// TwinCAT 3 PLC project MQPLC
// Title: YK_RFH
// Company: YK
// Author: SJ
// ProjectVersion: V1.1
// ProgramVersion: 3.1.4024.0
// CompilerDefines: VISU_USEWSTRING
// libraries:
//   Lib_Basic, * (Beckhoff_GZ)
//   Lib_FileOperation, * (Beckhoff_GZ)
//   Tc2_EtherCAT, * (Beckhoff Automation GmbH)
//   Tc2_Math, * (Beckhoff Automation GmbH)
//   Tc2_MC2, * (Beckhoff Automation GmbH)
//   Tc2_MC2_Camming, * (Beckhoff Automation GmbH)
//   Tc2_MC2_FlyingSaw, * (Beckhoff Automation GmbH)
//   Tc2_Standard, * (Beckhoff Automation GmbH)
//   Tc2_System, * (Beckhoff Automation GmbH)
//   Tc2_TcpIp, * (Beckhoff Automation GmbH)
//   Tc2_Utilities, * (Beckhoff Automation GmbH)
//   Tc2_XmlDataSrv, * (Beckhoff Automation GmbH)
//   Tc3_MC2_AdvancedHoming, * (Beckhoff Automation GmbH)
//   Tc3_Module, * (Beckhoff Automation GmbH)
//   VisuDialogs, * (System)
//   VisuElemEventTable, * (System)
//   VisuSymbols, * (System)
//   VisuSymbols,3.5.10.0,System
// project tree:
//   DUTs/01_AxisCO_Ntrol/ ST_ECYCtrl.TcDUT, ST_JXCE.TcDUT, ST_DustMotor.TcDUT, MC_AxisParameter.TcDUT, ST_SetpMotor.TcDUT
//   DUTs/01_AxisCO_Ntrol_1/ ST_AxisCmd.TcDUT, ST_AxisCtrl.TcDUT, ST_AxisIo.TcDUT, ST_AxisStatus.TcDUT, ST_Axis_Par.TcDUT
//   DUTs/02_Cylinder/ ST_CyCmd.TcDUT, ST_CyCtrl.TcDUT, ST_CYIo.TcDUT, ST_CyStatus.TcDUT
//   DUTs/04_Rectify/ ST_RecCtrl.TcDUT, ST_RecCmd.TcDUT, ST_RecIo.TcDUT, ST_RecStatus.TcDUT
//   DUTs/06_Interface/FB_Interface/ ST_Cam.TcDUT, ST_Gear.TcDUT, ST_GearInPos.TcDUT, ST_RecY.TcDUT, ST_TenBuffer.TcDUT, ST_Tension_1.TcDUT, ST_Tension.TcDUT
//   DUTs/06_Interface/Method/ ST_Method.TcDUT, ST_MethodOut.TcDUT
//   DUTs/07_Name/ ST_MotorName.TcDUT, ST_NGMark.TcDUT, ST_TableNo.TcDUT, ST_CylinderName.TcDUT, ST_VirAxisName.TcDUT, ST_AxisName.TcDUT, ST_RecName.TcDUT, ST_ElectValveName.TcDUT
//   DUTs/09_保持型汇总/ LocalProduction.TcDUT, ST_Data.TcDUT, ST_Name.TcDUT, ST_Parameter.TcDUT
//   DUTs/30_Parameter/ ST_DT_To_MQ_MES.TcDUT, ST_MouldRecY.TcDUT, ST_MQ_To_DT_MES.TcDUT, ST_ParFilterAD.TcDUT, ST_ParFilterDA.TcDUT, ST_ParMachine.TcDUT, ST_MoQiePar.TcDUT, ST_ParProduct.TcDUT, ST_ParPublic.TcDUT, ST_ParTemperature.TcDUT
//   DUTs/31_其他辅助/ ST_Timedata_2.TcDUT, File_com_typ.TcDUT, ST_DATA_NEED_BE_PERSIS.TcDUT
//   DUTs/32_系统/ ST_SystemPart.TcDUT, IModeEN.TcDUT, IRecipe.TcDUT, ST_SysCmd.TcDUT, ST_SystemPublic.TcDUT
//   DUTs/33_M2/ ST_BeltData.TcDUT, ST_TabData.TcDUT, ST_AlarmWarn.TcDUT, ST_BeltNo.TcDUT, ST_IntervalData.TcDUT, ST_IntervalNo.TcDUT, ST_TabNo.TcDUT
//   DUTs/34_M1/ ST_CCDio.TcDUT, ST_Rectify.TcDUT
//   DUTs/35_CCD/ ST_CCDComCuter.TcDUT, ST_CCDComLineScan.TcDUT, ST_CCDComR_Mould.TcDUT, ST_CCDComSize.TcDUT, ST_CCDCom.TcDUT, STCcdData.TcDUT, STCcdDataSend.TcDUT
//   DUTs/38_交互/ DToM_Process.TcDUT, DToM_System.TcDUT, MToD_Process.TcDUT, MToD_System.TcDUT, ST_P2InteractPart.TcDUT, ST_P2InteractPub.TcDUT
//   DUTs/39_记忆/ ST_Meney_Type.TcDUT
//   DUTs/MES/ DTM_Mes1.TcDUT, MTD_Mes1.TcDUT
//   DUTs/指纹/ ST_FingerprintKey.TcDUT
//   GVLs/ GVL_Par.TcGVL, GVL_Rectify.TcGVL, GVL_User2.TcGVL, GVL_User3.TcGVL, GCylinder.TcGVL, IO.TcGVL, GMotion.TcGVL, N.TcGVL, System.TcGVL, User01.TcGVL
//   POUs/BasicFunction/Basic/01_IO/ FB_Filter_AD.TcPOU (encrypted, skipped), FB_Filter_ADV2.TcPOU, FB_RotateSwitchCode.TcPOU (encrypted, skipped)
//   POUs/BasicFunction/Basic/02_Temperature/ FB_Blink.TcPOU (encrypted, skipped), FB_PulsPercentage.TcPOU (encrypted, skipped)
//   POUs/BasicFunction/Basic/03_Motion/ CS_AxisCtrl.TcPOU (encrypted, skipped)
//   POUs/BasicFunction/Basic/04_Gear/ FB_GearInDyn.TcPOU (encrypted, skipped), FB_GearInMulti.TcPOU (encrypted, skipped), FB_GearInPos.TcPOU (encrypted, skipped)
//   POUs/BasicFunction/Basic/05_Actuators/ FB_CylinderV2.TcPOU
//   POUs/BasicFunction/Basic/06_Public/ FC_AngleToLength.TcPOU (encrypted, skipped), FC_LengthToAngle.TcPOU (encrypted, skipped), f_Length2.TcPOU (encrypted, skipped), f_Length2_1.TcPOU (encrypted, skipped), PulseCtrl.TcPOU (encrypted, skipped), PulseGeneratorCtrl.TcPOU (encrypted, skipped)
//   POUs/BasicFunction/Basic/07_Ten/ FB_TensionBuffer.TcPOU (encrypted, skipped), FB_TensionPole.TcPOU, FB_TensionV3.TcPOU (encrypted, skipped), FB_TensionVirDriver.TcPOU
//   POUs/BasicFunction/Data/ Day_date.TcPOU, FB_DataTime.TcPOU, FB_ProductionDataLocal.TcPOU, FC_Filter_AA.TcPOU, FC_Variance.TcPOU, ScaleTrans.TcPOU, CS_Data.TcPOU, CS_Data_Test.TcPOU, CS_Recipe.TcPOU
//   POUs/BasicFunction/Motion/ Ax_FindHomeV3.TcPOU (encrypted, skipped), CS_DustMoter.TcPOU, FB_Electric_CY.TcPOU, FB_RectifyGM.TcPOU (encrypted, skipped), FB_TailCurl_PID.TcPOU, MS_Alarm.TcPOU, CS_SetpMoter.TcPOU
//   POUs/BasicFunction/User1/ FB_CamMQBeltV1.TcPOU (encrypted, skipped), FB_CamMQCCDPressV1.TcPOU (encrypted, skipped), FB_CamMQDriverV1.TcPOU (encrypted, skipped), FB_CamMQPushV1.TcPOU (encrypted, skipped), FB_CamMQPushV2.TcPOU (encrypted, skipped), FB_CamPoleBuffer.TcPOU (encrypted, skipped), FB_CamPoleBufferV2.TcPOU (encrypted, skipped), FB_CamPoleBuffer_1.TcPOU (encrypted, skipped), FB_CamPoleBuffer_BAK.TcPOU (encrypted, skipped), FB_CamVirDriver.TcPOU (encrypted, skipped), FB_CCD_Rounde.TcPOU, FB_DataXML.TcPOU, FB_DataXML_Old.TcPOU, FB_Rectify.TcPOU (encrypted, skipped), FB_TensionPole_1.TcPOU (encrypted, skipped)
//   POUs/BasicFunction/XFC/ FB_EL1259_IN.TcPOU, FB_TouchProbe_Ear.TcPOU
//   DUTs/08_IO/ ST_MoQieSenser.TcDUT, ST_MoQieButton.TcDUT
//   DUTs/06_Interface/ IData.TcDUT, IM2Glue.TcDUT
//   DUTs/36_ShortTest/ CMD.TcDUT, IShortTest.TcDUT, ShortDataShow.TcDUT, ShortPar.TcDUT
//   DUTs/37_Code/ ICode.TcDUT
//   POUs/BasicFunction/MES/ CS_CcdTcp.TcPOU, CS_CcdTcp_V2.TcPOU, CS_CodeTcp.TcPOU
//   POUs/BasicFunction/SystemInfo/ SystemInfoCtrl.TcPOU, TaskInfoCtrl.TcPOU
//   POUs/POUs/ AnPart.TcPOU, CaPart.TcPOU, FB_UserMain.TcPOU, FingerprintKey.TcPOU, IOLink.TcPOU, MAIN.TcPOU, MainState.TcPOU, ProductLocal.TcPOU
//   / Task_P1.TcTTO
// (motion and I/O tree: see PLC project dpplc)
// real-time tasks:
//   TASK Task P1: cycle T#2ms, priority 8, ADS port 350
//   TASK Task P2M1: cycle T#2ms, priority 16, ADS port 351
//   TASK Task P3: cycle T#2ms, priority 18, ADS port 352
//   TASK Task P2M2: cycle T#2ms, priority 14, ADS port 353
//   TASK Task P2M3: cycle T#2ms, priority 12, ADS port 354
//   TASK Task P2Main: cycle T#2ms, priority 10, ADS port 355
// variable links:
//   DPPLC/DPPLC Instance <-> MQPLC/MQPLC Instance
//     Task_P2M3 Inputs/IO.M_Pro <-> Task_P1 Outputs/IO.M_Pro
//     Task_P2M3 Outputs/IO.D_Pro <-> Task_P1 Inputs/IO.D_Pro
//     Task_P2M3 Outputs/IO.D_Sys/P3ReadParDone <-> Task_P1 Inputs/IO.D_Sys/P3ReadParDone
//     Task_P2M3 Outputs/IO.D_Sys/P3SaveParDone <-> Task_P1 Inputs/IO.D_Sys/P3SaveParDone
//     Task_P2M3 Outputs/IO.D_Sys/bP2ClearDo <-> Task_P1 Inputs/IO.D_Sys/bP2ClearDo
//     Task_P2M3 Outputs/IO.D_Sys/bP2ClearDone <-> Task_P1 Inputs/IO.D_Sys/bP2ClearDone
//     Task_P2M3 Outputs/IO.D_Sys/bP2Estop <-> Task_P1 Inputs/IO.D_Sys/bP2Estop
//     Task_P2M3 Outputs/IO.D_Sys/bP2M1Enable <-> Task_P1 Inputs/IO.D_Sys/bP2M1Enable
//     Task_P2M3 Outputs/IO.D_Sys/bP2M2Enable <-> Task_P1 Inputs/IO.D_Sys/bP2M2Enable
//     Task_P2M3 Outputs/IO.D_Sys/bP2M3Enable <-> Task_P1 Inputs/IO.D_Sys/bP2M3Enable
//     Task_P2M3 Outputs/IO.D_Sys/bP2Runing <-> Task_P1 Inputs/IO.D_Sys/bP2Runing
//     Task_P2M3 Outputs/IO.D_Sys/bP2Start <-> Task_P1 Inputs/IO.D_Sys/bP2Start
//     Task_P2M3 Outputs/IO.D_Sys/fM1MainSetPos <-> Task_P1 Inputs/IO.D_Sys/fM1MainSetPos
//     Task_P2M3 Outputs/IO.D_Sys/fM2MainSetPos <-> Task_P1 Inputs/IO.D_Sys/fM2MainSetPos
//     Task_P2M3 Outputs/IO.D_Sys/fM3MainSetPos <-> Task_P1 Inputs/IO.D_Sys/fM3MainSetPos
//     Task_P2M3 Outputs/IO.D_Sys/iAn1Ask <-> Task_P1 Inputs/IO.D_Sys/iAn1Ask
//     Task_P2M3 Outputs/IO.D_Sys/iAn2Ask <-> Task_P1 Inputs/IO.D_Sys/iAn2Ask
//     Task_P2M3 Outputs/IO.D_Sys/iAn3Ask <-> Task_P1 Inputs/IO.D_Sys/iAn3Ask
//     Task_P2M3 Outputs/IO.D_Sys/iCa1Ask <-> Task_P1 Inputs/IO.D_Sys/iCa1Ask
//     Task_P2M3 Outputs/IO.D_Sys/iCa2Ask <-> Task_P1 Inputs/IO.D_Sys/iCa2Ask
//     Task_P2M3 Outputs/IO.D_Sys/iCa3Ask <-> Task_P1 Inputs/IO.D_Sys/iCa3Ask
//     Task_P2Main Inputs/IO.AnMQ_MES1 <-> Task_P1 Outputs/IO.AnMQ_MES1
//     Task_P2Main Inputs/IO.AnMQ_MES2 <-> Task_P1 Outputs/IO.AnMQ_MES2
//     Task_P2Main Inputs/IO.AnMQ_MES3 <-> Task_P1 Outputs/IO.AnMQ_MES3
//     Task_P2Main Inputs/IO.CaMQ_MES1 <-> Task_P1 Outputs/IO.CaMQ_MES1
//     Task_P2Main Inputs/IO.CaMQ_MES2 <-> Task_P1 Outputs/IO.CaMQ_MES2
//     Task_P2Main Inputs/IO.CaMQ_MES3 <-> Task_P1 Outputs/IO.CaMQ_MES3
//     Task_P2Main Outputs/IO.YL_Q <-> Task_P1 Inputs/IO.YL_I
//     Task_P3 Inputs/IO.M_Sys/P1ReadParDone <-> Task_P1 Outputs/IO.M_Sys/P1ReadParDone
//     Task_P3 Inputs/IO.M_Sys/P1SaveParDone <-> Task_P1 Outputs/IO.M_Sys/P1SaveParDone
//     Task_P3 Inputs/IO.M_Sys/bP1ClearDo <-> Task_P1 Outputs/IO.M_Sys/bP1ClearDo
//     Task_P3 Inputs/IO.M_Sys/bP1ClearDone <-> Task_P1 Outputs/IO.M_Sys/bP1ClearDone
//     Task_P3 Inputs/IO.M_Sys/bP1Estop <-> Task_P1 Outputs/IO.M_Sys/bP1Estop
//     Task_P3 Inputs/IO.M_Sys/bP1Runing <-> Task_P1 Outputs/IO.M_Sys/bP1Runing
//     Task_P3 Inputs/IO.M_Sys/bP1Start <-> Task_P1 Outputs/IO.M_Sys/bP1Start
//     Task_P3 Inputs/IO.M_Sys/iCarryPoleMode <-> Task_P1 Outputs/IO.M_Sys/iCarryPoleMode
//     Task_P3 Inputs/IO.M_Sys/p1state <-> Task_P1 Outputs/IO.M_Sys/p1state
//     Task_P3 Inputs/IO.YL_INT1 <-> Task_P1 Outputs/IO.YL_INT1
//     Task_P3 Inputs/P3IO.MTD_Mes1/bFuncEN <-> Task_P1 Outputs/IO.MTD_Mes1/bFuncEN
//     Task_P3 Inputs/P3IO.MTD_Mes1/rExcelRate <-> Task_P1 Outputs/IO.MTD_Mes1/rExcelRate
//     Task_P3 Inputs/P3IO.MTD_Mes1/uOther <-> Task_P1 Outputs/IO.MTD_Mes1/uOther
//     Task_P3 Inputs/P3Par.MQ_To_DT_MES <-> Task_P1 Outputs/IO.MQ_To_DT_MES
//     Task_P3 Outputs/IO.YL_INT2 <-> Task_P1 Inputs/IO.YL_INT2
//     Task_P3 Outputs/P3IO.DTM_Mes1/bFuncEN <-> Task_P1 Inputs/IO.DTM_Mes1/bFuncEN
//     Task_P3 Outputs/P3IO.DTM_Mes1/uOther <-> Task_P1 Inputs/IO.DTM_Mes1/uOther
//     Task_P3 Outputs/P3Par.DT_To_MQ_MES <-> Task_P1 Inputs/IO.DT_To_MQ_MES
//   MQPLC/MQPLC Instance <-> Device 3 (EtherCAT)/Box 2 (CU1128)/Term 24 (CU1128-B)/负极上表面除尘皮带(InoSV660N)
//     Task_P1 Inputs/GMotion.DrivesOP[42] <-> InfoData/State
//     Task_P1 Inputs/GMotion.arrAxisCtrl[42].Io.DigitalInputs <-> Inputs/Digital inputs
//     Task_P1 Inputs/GMotion.arrAxisCtrl[42].Io.ErrorCode <-> Inputs/Error code
//     Task_P1 Inputs/GMotion.iActTorque_M[42] <-> Inputs/Torque actual value
//   MQPLC/MQPLC Instance <-> Device 3 (EtherCAT)/Box 2 (CU1128)/Term 24 (CU1128-B)/负极下表面除尘倒装皮带(InoSV660N)
//     Task_P1 Inputs/GMotion.DrivesOP[43] <-> InfoData/State
//     Task_P1 Inputs/GMotion.arrAxisCtrl[43].Io.DigitalInputs <-> Inputs/Digital inputs
//     Task_P1 Inputs/GMotion.arrAxisCtrl[43].Io.ErrorCode <-> Inputs/Error code
//     Task_P1 Inputs/GMotion.iActTorque_M[43] <-> Inputs/Torque actual value
//   MQPLC/MQPLC Instance <-> Device 3 (EtherCAT)/Box 2 (CU1128)/Term 24 (CU1128-B)/负极倒角模具(InoSV660N)
//     Task_P1 Inputs/GMotion.DrivesOP[30] <-> InfoData/State
//     Task_P1 Inputs/GMotion.arrAxisCtrl[30].Io.DigitalInputs <-> Inputs/Digital inputs
//     Task_P1 Inputs/GMotion.arrAxisCtrl[30].Io.ErrorCode <-> Inputs/Error code
//     Task_P1 Inputs/GMotion.iActTorque_M[30] <-> Inputs/Torque actual value
//   MQPLC/MQPLC Instance <-> Device 3 (EtherCAT)/Box 2 (CU1128)/Term 24 (CU1128-B)/负极右放卷电机(InoSV660N)
//     Task_P1 Inputs/GMotion.DrivesOP[26] <-> InfoData/State
//     Task_P1 Inputs/GMotion.arrAxisCtrl[26].Io.DigitalInputs <-> Inputs/Digital inputs
//     Task_P1 Inputs/GMotion.arrAxisCtrl[26].Io.ErrorCode <-> Inputs/Error code
//     Task_P1 Inputs/GMotion.iActTorque_M[26] <-> Inputs/Torque actual value
//   MQPLC/MQPLC Instance <-> Device 3 (EtherCAT)/Box 2 (CU1128)/Term 24 (CU1128-B)/负极尺寸CCD压片升降(InoSV660N)
//     Task_P1 Inputs/GMotion.DrivesOP[38] <-> InfoData/State
//     Task_P1 Inputs/GMotion.arrAxisCtrl[38].Io.DigitalInputs <-> Inputs/Digital inputs
//     Task_P1 Inputs/GMotion.arrAxisCtrl[38].Io.ErrorCode <-> Inputs/Error code
//     Task_P1 Inputs/GMotion.iActTorque_M[38] <-> Inputs/Torque actual value
//   MQPLC/MQPLC Instance <-> Device 3 (EtherCAT)/Box 2 (CU1128)/Term 24 (CU1128-B)/负极左放卷电机(InoSV660N)
//     Task_P1 Inputs/GMotion.DrivesOP[25] <-> InfoData/State
//     Task_P1 Inputs/GMotion.arrAxisCtrl[25].Io.DigitalInputs <-> Inputs/Digital inputs
//     Task_P1 Inputs/GMotion.arrAxisCtrl[25].Io.ErrorCode <-> Inputs/Error code
//     Task_P1 Inputs/GMotion.iActTorque_M[25] <-> Inputs/Torque actual value
//   MQPLC/MQPLC Instance <-> Device 3 (EtherCAT)/Box 2 (CU1128)/Term 24 (CU1128-B)/负极模具纠偏X轴(肩宽)(InoSV660N)
//     Task_P1 Inputs/GMotion.DrivesOP[31] <-> InfoData/State
//     Task_P1 Inputs/GMotion.arrAxisCtrl[31].Io.DigitalInputs <-> Inputs/Digital inputs
//     Task_P1 Inputs/GMotion.arrAxisCtrl[31].Io.ErrorCode <-> Inputs/Error code
//     Task_P1 Inputs/GMotion.iActTorque_M[31] <-> Inputs/Torque actual value
//   MQPLC/MQPLC Instance <-> Device 3 (EtherCAT)/Box 2 (CU1128)/Term 24 (CU1128-B)/负极模具纠偏Y轴(InoSV660N)
//     Task_P1 Inputs/GMotion.DrivesOP[32] <-> InfoData/State
//     Task_P1 Inputs/GMotion.arrAxisCtrl[32].Io.DigitalInputs <-> Inputs/Digital inputs
//     Task_P1 Inputs/GMotion.arrAxisCtrl[32].Io.ErrorCode <-> Inputs/Error code
//     Task_P1 Inputs/GMotion.iActTorque_M[32] <-> Inputs/Torque actual value
//   MQPLC/MQPLC Instance <-> Device 3 (EtherCAT)/Box 2 (CU1128)/Term 24 (CU1128-B)/负极模切主驱动(CDHD)
//     Task_P1 Inputs/GMotion.DrivesOP[33] <-> InfoData/State
//     Task_P1 Inputs/GMotion.arrAxisCtrl[33].Io.DigitalInputs <-> TxPDO 4/Digital inputs
//     Task_P1 Inputs/GMotion.iActTorque_M[33] <-> TxPDO 1/Torque Actual Value
//   MQPLC/MQPLC Instance <-> Device 3 (EtherCAT)/Box 2 (CU1128)/Term 24 (CU1128-B)/负极模切前摆杆张力(InoSV660N)
//     Task_P1 Inputs/GMotion.DrivesOP[27] <-> InfoData/State
//     Task_P1 Inputs/GMotion.arrAxisCtrl[27].Io.DigitalInputs <-> Inputs/Digital inputs
//     Task_P1 Inputs/GMotion.arrAxisCtrl[27].Io.ErrorCode <-> Inputs/Error code
//     Task_P1 Inputs/GMotion.iActDriveTorque[2] <-> Inputs/Torque actual value
//     Task_P1 Outputs/GMotion.iMaxProfileVelo[2] <-> Outputs/Max profile velocity
//     Task_P1 Outputs/GMotion.iNegtiveTorqueLimits[2] <-> Outputs/Negative torque limit value
//     Task_P1 Outputs/GMotion.iPostiveTorqueLimits[2] <-> Outputs/Positive torque limit value
//     Task_P1 Outputs/GMotion.iSetDriveMode[2] <-> Outputs/Modes of operation
//     Task_P1 Outputs/GMotion.iTargetTorque[2] <-> Outputs/Target torque
//   MQPLC/MQPLC Instance <-> Device 3 (EtherCAT)/Box 2 (CU1128)/Term 24 (CU1128-B)/负极模切极片缓存(CDHD)
//     Task_P1 Inputs/GMotion.DrivesOP[29] <-> InfoData/State
//     Task_P1 Inputs/GMotion.arrAxisCtrl[29].Io.DigitalInputs <-> TxPDO 4/Digital inputs
//     Task_P1 Inputs/GMotion.iActTorque_M[29] <-> TxPDO 1/Torque Actual Value
//   MQPLC/MQPLC Instance <-> Device 3 (EtherCAT)/Box 2 (CU1128)/Term 24 (CU1128-B)/负极模切辅助驱动(InoSV660N)
//     Task_P1 Inputs/GMotion.DrivesOP[28] <-> InfoData/State
//     Task_P1 Inputs/GMotion.arrAxisCtrl[28].Io.DigitalInputs <-> Inputs/Digital inputs
//     Task_P1 Inputs/GMotion.arrAxisCtrl[28].Io.ErrorCode <-> Inputs/Error code
//     Task_P1 Inputs/GMotion.iActTorque_M[28] <-> Inputs/Torque actual value
//   MQPLC/MQPLC Instance <-> Device 3 (EtherCAT)/Box 2 (CU1128)/Term 24 (CU1128-B)/负极裁切切刀(InoSV660N)
//     Task_P1 Inputs/GMotion.DrivesOP[34] <-> InfoData/State
//     Task_P1 Inputs/GMotion.arrAxisCtrl[34].Io.DigitalInputs <-> Inputs/Digital inputs
//     Task_P1 Inputs/GMotion.arrAxisCtrl[34].Io.ErrorCode <-> Inputs/Error code
//     Task_P1 Inputs/GMotion.iActTorque_M[34] <-> Inputs/Torque actual value
//   MQPLC/MQPLC Instance <-> Device 3 (EtherCAT)/Box 2 (CU1128)/Term 24 (CU1128-B)/负极裁切角度纠偏(InoSV660N)
//     Task_P1 Inputs/GMotion.DrivesOP[35] <-> InfoData/State
//     Task_P1 Inputs/GMotion.arrAxisCtrl[35].Io.DigitalInputs <-> Inputs/Digital inputs
//     Task_P1 Inputs/GMotion.arrAxisCtrl[35].Io.ErrorCode <-> Inputs/Error code
//     Task_P1 Inputs/GMotion.iActTorque_M[35] <-> Inputs/Torque actual value
//   MQPLC/MQPLC Instance <-> Device 3 (EtherCAT)/Box 2 (CU1128)/Term 24 (CU1128-B)/负极裁切输送带换型(InoSV660N)
//     Task_P1 Inputs/GMotion.DrivesOP[37] <-> InfoData/State
//     Task_P1 Inputs/GMotion.arrAxisCtrl[37].Io.DigitalInputs <-> Inputs/Digital inputs
//     Task_P1 Inputs/GMotion.arrAxisCtrl[37].Io.ErrorCode <-> Inputs/Error code
//     Task_P1 Inputs/GMotion.iActTorque_M[37] <-> Inputs/Torque actual value
//   MQPLC/MQPLC Instance <-> Device 3 (EtherCAT)/Box 2 (CU1128)/Term 24 (CU1128-B)/负极裁切输送皮带(InoSV660N)
//     Task_P1 Inputs/GMotion.DrivesOP[36] <-> InfoData/State
//     Task_P1 Inputs/GMotion.arrAxisCtrl[36].Io.DigitalInputs <-> Inputs/Digital inputs
//     Task_P1 Inputs/GMotion.arrAxisCtrl[36].Io.ErrorCode <-> Inputs/Error code
//     Task_P1 Inputs/GMotion.iActTorque_M[36] <-> Inputs/Torque actual value
//   MQPLC/MQPLC Instance <-> Device 3 (EtherCAT)/Box 2 (CU1128)/Term 24 (CU1128-B)/负极踢单张废料(InoSV660N)
//     Task_P1 Inputs/GMotion.DrivesOP[41] <-> InfoData/State
//     Task_P1 Inputs/GMotion.arrAxisCtrl[41].Io.DigitalInputs <-> Inputs/Digital inputs
//     Task_P1 Inputs/GMotion.arrAxisCtrl[41].Io.ErrorCode <-> Inputs/Error code
//     Task_P1 Inputs/GMotion.iActTorque_M[41] <-> Inputs/Torque actual value
//   MQPLC/MQPLC Instance <-> Device 3 (EtherCAT)/Box 2 (CU1128)/Term 24 (CU1128-B)/负极踢废倒装皮带(InoSV660N)
//     Task_P1 Inputs/GMotion.DrivesOP[39] <-> InfoData/State
//     Task_P1 Inputs/GMotion.arrAxisCtrl[39].Io.DigitalInputs <-> Inputs/Digital inputs
//     Task_P1 Inputs/GMotion.arrAxisCtrl[39].Io.ErrorCode <-> Inputs/Error code
//     Task_P1 Inputs/GMotion.iActTorque_M[39] <-> Inputs/Torque actual value
//   MQPLC/MQPLC Instance <-> Device 3 (EtherCAT)/Box 2 (CU1128)/Term 24 (CU1128-B)/负极踢连续废料(InoSV660N)
//     Task_P1 Inputs/GMotion.DrivesOP[40] <-> InfoData/State
//     Task_P1 Inputs/GMotion.arrAxisCtrl[40].Io.DigitalInputs <-> Inputs/Digital inputs
//     Task_P1 Inputs/GMotion.arrAxisCtrl[40].Io.ErrorCode <-> Inputs/Error code
//     Task_P1 Inputs/GMotion.iActTorque_M[40] <-> Inputs/Torque actual value
//   MQPLC/MQPLC Instance <-> Device 3 (EtherCAT)/Box 2 (CU1128)/Term 44 (CU1128-C)/P2M2正极送料分段皮带2[21(模切)] (InoSV660N)
//     Task_P1 Inputs/GMotion.arrAxisCtrl[21].Io.ErrorCode <-> Inputs/Error code
//     Task_P1 Inputs/GMotion.iActTorque_M[21] <-> Inputs/Torque actual value
//   MQPLC/MQPLC Instance <-> Device 3 (EtherCAT)/Box 2 (CU1128)/Term 44 (CU1128-C)/P2M2负极送料分段皮带2（45模切） (InoSV660N)
//     Task_P1 Inputs/GMotion.arrAxisCtrl[45].Io.ErrorCode <-> Inputs/Error code
//     Task_P1 Inputs/GMotion.iActTorque_M[45] <-> Inputs/Torque actual value
//   MQPLC/MQPLC Instance <-> Device 3 (EtherCAT)/Box 2 (CU1128)/Term 44 (CU1128-C)/P2M3正极送料分段皮带3（22模切） (InoSV660N)
//     Task_P1 Inputs/GMotion.arrAxisCtrl[22].Io.ErrorCode <-> Inputs/Error code
//     Task_P1 Inputs/GMotion.iActTorque_M[22] <-> Inputs/Torque actual value
//   MQPLC/MQPLC Instance <-> Device 3 (EtherCAT)/Box 2 (CU1128)/Term 44 (CU1128-C)/P2M3负极送料分段皮带3（46模切） (InoSV660N)
//     Task_P1 Inputs/GMotion.arrAxisCtrl[46].Io.ErrorCode <-> Inputs/Error code
//     Task_P1 Inputs/GMotion.iActTorque_M[46] <-> Inputs/Torque actual value
//   MQPLC/MQPLC Instance <-> Device 3 (EtherCAT)/Box 2 (CU1128)/一号叠片IO耦合器(GSIO-A-ECC)
//     Task_P1 Inputs/IO.I30101 <-> I301/Digital Inputs/Channel 1
//     Task_P1 Inputs/IO.I30107 <-> I301/Digital Inputs/Channel 7
//     Task_P1 Outputs/IO.Q30103 <-> Q301/Digital Outputs/Channel 3
//     Task_P1 Outputs/IO.Q30104 <-> Q301/Digital Outputs/Channel 4
//     Task_P1 Outputs/IO.Q30201 <-> Q302/Digital Outputs/Channel 1
//     Task_P1 Outputs/IO.Q30202 <-> Q302/Digital Outputs/Channel 2
//   MQPLC/MQPLC Instance <-> Device 3 (EtherCAT)/Box 2 (CU1128)/三号叠片IO耦合器(GSIO-A-ECC)
//     Task_P1 Inputs/IO.I50101 <-> I501 (GSIO-A-16DIN)/Digital Inputs/Channel 1
//     Task_P1 Inputs/IO.I50107 <-> I501 (GSIO-A-16DIN)/Digital Inputs/Channel 7
//     Task_P1 Outputs/IO.Q50103 <-> Q501 (GSIO-A-16DON)/Digital Outputs/Channel 3
//     Task_P1 Outputs/IO.Q50104 <-> Q501 (GSIO-A-16DON)/Digital Outputs/Channel 4
//     Task_P1 Outputs/IO.Q50201 <-> Q502 (GSIO-A-16DON)/Digital Outputs/Channel 1
//     Task_P1 Outputs/IO.Q50202 <-> Q502 (GSIO-A-16DON)/Digital Outputs/Channel 2
//   MQPLC/MQPLC Instance <-> Device 3 (EtherCAT)/Box 2 (CU1128)/二号叠片IO耦合器 (GSIO-A-ECC)
//     Task_P1 Inputs/IO.I40101 <-> I401 (GSIO-A-16DIN)/Digital Inputs/Channel 1
//     Task_P1 Inputs/IO.I40107 <-> I401 (GSIO-A-16DIN)/Digital Inputs/Channel 7
//     Task_P1 Outputs/IO.Q40103 <-> O401 (GSIO-A-16DON)/Digital Outputs/Channel 3
//     Task_P1 Outputs/IO.Q40104 <-> O401 (GSIO-A-16DON)/Digital Outputs/Channel 4
//     Task_P1 Outputs/IO.Q40201 <-> O402 (GSIO-A-16DON)/Digital Outputs/Channel 1
//     Task_P1 Outputs/IO.Q40202 <-> O402 (GSIO-A-16DON)/Digital Outputs/Channel 2
//   MQPLC/MQPLC Instance <-> Device 3 (EtherCAT)/Box 2 (CU1128)/正极IO耦合器(GSIO-A-ECC)
//     Task_P1 Inputs/IO.AI101[0] <-> AI101 (GSIO-A-4AIHV)/Analog Inputs/Channel 1
//     Task_P1 Inputs/IO.AI101[1] <-> AI101 (GSIO-A-4AIHV)/Analog Inputs/Channel 2
//     Task_P1 Inputs/IO.AI101[2] <-> AI101 (GSIO-A-4AIHV)/Analog Inputs/Channel 3
//     Task_P1 Inputs/IO.AI101[3] <-> AI101 (GSIO-A-4AIHV)/Analog Inputs/Channel 4
//     Task_P1 Inputs/IO.AI102[0] <-> AI102 (GSIO-A-4AIHV)/Analog Inputs/Channel 1
//     Task_P1 Inputs/IO.AI102[1] <-> AI102 (GSIO-A-4AIHV)/Analog Inputs/Channel 2
//     Task_P1 Inputs/IO.AI102[2] <-> AI102 (GSIO-A-4AIHV)/Analog Inputs/Channel 3
//     Task_P1 Inputs/IO.AI102[3] <-> AI102 (GSIO-A-4AIHV)/Analog Inputs/Channel 4
//     Task_P1 Inputs/IO.I101[10] <-> I101 (GSIO-A-16DIN)/Digital Inputs/Channel 10
//     Task_P1 Inputs/IO.I101[11] <-> I101 (GSIO-A-16DIN)/Digital Inputs/Channel 11
//     Task_P1 Inputs/IO.I101[12] <-> I101 (GSIO-A-16DIN)/Digital Inputs/Channel 12
//     Task_P1 Inputs/IO.I101[13] <-> I101 (GSIO-A-16DIN)/Digital Inputs/Channel 13
//     Task_P1 Inputs/IO.I101[14] <-> I101 (GSIO-A-16DIN)/Digital Inputs/Channel 14
//     Task_P1 Inputs/IO.I101[15] <-> I101 (GSIO-A-16DIN)/Digital Inputs/Channel 15
//     Task_P1 Inputs/IO.I101[16] <-> I101 (GSIO-A-16DIN)/Digital Inputs/Channel 16
//     Task_P1 Inputs/IO.I101[1] <-> I101 (GSIO-A-16DIN)/Digital Inputs/Channel 1
//     Task_P1 Inputs/IO.I101[2] <-> I101 (GSIO-A-16DIN)/Digital Inputs/Channel 2
//     Task_P1 Inputs/IO.I101[3] <-> I101 (GSIO-A-16DIN)/Digital Inputs/Channel 3
//     Task_P1 Inputs/IO.I101[4] <-> I101 (GSIO-A-16DIN)/Digital Inputs/Channel 4
//     Task_P1 Inputs/IO.I101[5] <-> I101 (GSIO-A-16DIN)/Digital Inputs/Channel 5
//     Task_P1 Inputs/IO.I101[6] <-> I101 (GSIO-A-16DIN)/Digital Inputs/Channel 6
//     Task_P1 Inputs/IO.I101[7] <-> I101 (GSIO-A-16DIN)/Digital Inputs/Channel 7
//     Task_P1 Inputs/IO.I101[8] <-> I101 (GSIO-A-16DIN)/Digital Inputs/Channel 8
//     Task_P1 Inputs/IO.I101[9] <-> I101 (GSIO-A-16DIN)/Digital Inputs/Channel 9
//     Task_P1 Inputs/IO.I102[10] <-> I102 (GSIO-A-16DIN)/Digital Inputs/Channel 10
//     Task_P1 Inputs/IO.I102[11] <-> I102 (GSIO-A-16DIN)/Digital Inputs/Channel 11
//     Task_P1 Inputs/IO.I102[12] <-> I102 (GSIO-A-16DIN)/Digital Inputs/Channel 12
//     Task_P1 Inputs/IO.I102[13] <-> I102 (GSIO-A-16DIN)/Digital Inputs/Channel 13
//     Task_P1 Inputs/IO.I102[14] <-> I102 (GSIO-A-16DIN)/Digital Inputs/Channel 14
//     Task_P1 Inputs/IO.I102[15] <-> I102 (GSIO-A-16DIN)/Digital Inputs/Channel 15
//     Task_P1 Inputs/IO.I102[16] <-> I102 (GSIO-A-16DIN)/Digital Inputs/Channel 16
//     Task_P1 Inputs/IO.I102[1] <-> I102 (GSIO-A-16DIN)/Digital Inputs/Channel 1
//     Task_P1 Inputs/IO.I102[2] <-> I102 (GSIO-A-16DIN)/Digital Inputs/Channel 2
//     Task_P1 Inputs/IO.I102[3] <-> I102 (GSIO-A-16DIN)/Digital Inputs/Channel 3
//     Task_P1 Inputs/IO.I102[4] <-> I102 (GSIO-A-16DIN)/Digital Inputs/Channel 4
//     Task_P1 Inputs/IO.I102[5] <-> I102 (GSIO-A-16DIN)/Digital Inputs/Channel 5
//     Task_P1 Inputs/IO.I102[6] <-> I102 (GSIO-A-16DIN)/Digital Inputs/Channel 6
//     Task_P1 Inputs/IO.I102[7] <-> I102 (GSIO-A-16DIN)/Digital Inputs/Channel 7
//     Task_P1 Inputs/IO.I102[8] <-> I102 (GSIO-A-16DIN)/Digital Inputs/Channel 8
//     Task_P1 Inputs/IO.I102[9] <-> I102 (GSIO-A-16DIN)/Digital Inputs/Channel 9
//     Task_P1 Inputs/IO.I103[10] <-> I103 (GSIO-A-16DIN)/Digital Inputs/Channel 10
//     Task_P1 Inputs/IO.I103[11] <-> I103 (GSIO-A-16DIN)/Digital Inputs/Channel 11
//     Task_P1 Inputs/IO.I103[12] <-> I103 (GSIO-A-16DIN)/Digital Inputs/Channel 12
//     Task_P1 Inputs/IO.I103[13] <-> I103 (GSIO-A-16DIN)/Digital Inputs/Channel 13
//     Task_P1 Inputs/IO.I103[14] <-> I103 (GSIO-A-16DIN)/Digital Inputs/Channel 14
//     Task_P1 Inputs/IO.I103[15] <-> I103 (GSIO-A-16DIN)/Digital Inputs/Channel 15
//     Task_P1 Inputs/IO.I103[16] <-> I103 (GSIO-A-16DIN)/Digital Inputs/Channel 16
//     Task_P1 Inputs/IO.I103[1] <-> I103 (GSIO-A-16DIN)/Digital Inputs/Channel 1
//     Task_P1 Inputs/IO.I103[2] <-> I103 (GSIO-A-16DIN)/Digital Inputs/Channel 2
//     Task_P1 Inputs/IO.I103[3] <-> I103 (GSIO-A-16DIN)/Digital Inputs/Channel 3
//     Task_P1 Inputs/IO.I103[4] <-> I103 (GSIO-A-16DIN)/Digital Inputs/Channel 4
//     Task_P1 Inputs/IO.I103[5] <-> I103 (GSIO-A-16DIN)/Digital Inputs/Channel 5
//     Task_P1 Inputs/IO.I103[6] <-> I103 (GSIO-A-16DIN)/Digital Inputs/Channel 6
//     Task_P1 Inputs/IO.I103[7] <-> I103 (GSIO-A-16DIN)/Digital Inputs/Channel 7
//     Task_P1 Inputs/IO.I103[8] <-> I103 (GSIO-A-16DIN)/Digital Inputs/Channel 8
//     Task_P1 Inputs/IO.I103[9] <-> I103 (GSIO-A-16DIN)/Digital Inputs/Channel 9
//     Task_P1 Inputs/IO.I104[10] <-> I104 (GSIO-A-16DIN)/Digital Inputs/Channel 10
//     Task_P1 Inputs/IO.I104[11] <-> I104 (GSIO-A-16DIN)/Digital Inputs/Channel 11
//     Task_P1 Inputs/IO.I104[12] <-> I104 (GSIO-A-16DIN)/Digital Inputs/Channel 12
//     Task_P1 Inputs/IO.I104[13] <-> I104 (GSIO-A-16DIN)/Digital Inputs/Channel 13
//     Task_P1 Inputs/IO.I104[14] <-> I104 (GSIO-A-16DIN)/Digital Inputs/Channel 14
//     Task_P1 Inputs/IO.I104[15] <-> I104 (GSIO-A-16DIN)/Digital Inputs/Channel 15
//     Task_P1 Inputs/IO.I104[16] <-> I104 (GSIO-A-16DIN)/Digital Inputs/Channel 16
//     Task_P1 Inputs/IO.I104[1] <-> I104 (GSIO-A-16DIN)/Digital Inputs/Channel 1
//     Task_P1 Inputs/IO.I104[2] <-> I104 (GSIO-A-16DIN)/Digital Inputs/Channel 2
//     Task_P1 Inputs/IO.I104[3] <-> I104 (GSIO-A-16DIN)/Digital Inputs/Channel 3
//     Task_P1 Inputs/IO.I104[4] <-> I104 (GSIO-A-16DIN)/Digital Inputs/Channel 4
//     Task_P1 Inputs/IO.I104[5] <-> I104 (GSIO-A-16DIN)/Digital Inputs/Channel 5
//     Task_P1 Inputs/IO.I104[6] <-> I104 (GSIO-A-16DIN)/Digital Inputs/Channel 6
//     Task_P1 Inputs/IO.I104[7] <-> I104 (GSIO-A-16DIN)/Digital Inputs/Channel 7
//     Task_P1 Inputs/IO.I104[8] <-> I104 (GSIO-A-16DIN)/Digital Inputs/Channel 8
//     Task_P1 Inputs/IO.I104[9] <-> I104 (GSIO-A-16DIN)/Digital Inputs/Channel 9
//     Task_P1 Inputs/IO.I105[10] <-> I105 (GSIO-A-16DIN)/Digital Inputs/Channel 10
//     Task_P1 Inputs/IO.I105[11] <-> I105 (GSIO-A-16DIN)/Digital Inputs/Channel 11
//     Task_P1 Inputs/IO.I105[12] <-> I105 (GSIO-A-16DIN)/Digital Inputs/Channel 12
//     Task_P1 Inputs/IO.I105[13] <-> I105 (GSIO-A-16DIN)/Digital Inputs/Channel 13
//     Task_P1 Inputs/IO.I105[14] <-> I105 (GSIO-A-16DIN)/Digital Inputs/Channel 14
//     Task_P1 Inputs/IO.I105[15] <-> I105 (GSIO-A-16DIN)/Digital Inputs/Channel 15
//     Task_P1 Inputs/IO.I105[16] <-> I105 (GSIO-A-16DIN)/Digital Inputs/Channel 16
//     Task_P1 Inputs/IO.I105[1] <-> I105 (GSIO-A-16DIN)/Digital Inputs/Channel 1
//     Task_P1 Inputs/IO.I105[2] <-> I105 (GSIO-A-16DIN)/Digital Inputs/Channel 2
//     Task_P1 Inputs/IO.I105[3] <-> I105 (GSIO-A-16DIN)/Digital Inputs/Channel 3
//     Task_P1 Inputs/IO.I105[4] <-> I105 (GSIO-A-16DIN)/Digital Inputs/Channel 4
//     Task_P1 Inputs/IO.I105[5] <-> I105 (GSIO-A-16DIN)/Digital Inputs/Channel 5
//     Task_P1 Inputs/IO.I105[6] <-> I105 (GSIO-A-16DIN)/Digital Inputs/Channel 6
//     Task_P1 Inputs/IO.I105[7] <-> I105 (GSIO-A-16DIN)/Digital Inputs/Channel 7
//     Task_P1 Inputs/IO.I105[8] <-> I105 (GSIO-A-16DIN)/Digital Inputs/Channel 8
//     Task_P1 Inputs/IO.I105[9] <-> I105 (GSIO-A-16DIN)/Digital Inputs/Channel 9
//     Task_P1 Inputs/IO.I106[10] <-> I106 (GSIO-A-16DIN)/Digital Inputs/Channel 10
//     Task_P1 Inputs/IO.I106[11] <-> I106 (GSIO-A-16DIN)/Digital Inputs/Channel 11
//     Task_P1 Inputs/IO.I106[12] <-> I106 (GSIO-A-16DIN)/Digital Inputs/Channel 12
//     Task_P1 Inputs/IO.I106[13] <-> I106 (GSIO-A-16DIN)/Digital Inputs/Channel 13
//     Task_P1 Inputs/IO.I106[14] <-> I106 (GSIO-A-16DIN)/Digital Inputs/Channel 14
//     Task_P1 Inputs/IO.I106[15] <-> I106 (GSIO-A-16DIN)/Digital Inputs/Channel 15
//     Task_P1 Inputs/IO.I106[16] <-> I106 (GSIO-A-16DIN)/Digital Inputs/Channel 16
//     Task_P1 Inputs/IO.I106[1] <-> I106 (GSIO-A-16DIN)/Digital Inputs/Channel 1
//     Task_P1 Inputs/IO.I106[2] <-> I106 (GSIO-A-16DIN)/Digital Inputs/Channel 2
//     Task_P1 Inputs/IO.I106[3] <-> I106 (GSIO-A-16DIN)/Digital Inputs/Channel 3
//     Task_P1 Inputs/IO.I106[4] <-> I106 (GSIO-A-16DIN)/Digital Inputs/Channel 4
//     Task_P1 Inputs/IO.I106[5] <-> I106 (GSIO-A-16DIN)/Digital Inputs/Channel 5
//     Task_P1 Inputs/IO.I106[6] <-> I106 (GSIO-A-16DIN)/Digital Inputs/Channel 6
//     Task_P1 Inputs/IO.I106[7] <-> I106 (GSIO-A-16DIN)/Digital Inputs/Channel 7
//     Task_P1 Inputs/IO.I106[8] <-> I106 (GSIO-A-16DIN)/Digital Inputs/Channel 8
//     Task_P1 Inputs/IO.I106[9] <-> I106 (GSIO-A-16DIN)/Digital Inputs/Channel 9
//     Task_P1 Inputs/IO.I107[10] <-> I107 (GSIO-A-16DIN)/Digital Inputs/Channel 10
//     Task_P1 Inputs/IO.I107[11] <-> I107 (GSIO-A-16DIN)/Digital Inputs/Channel 11
//     Task_P1 Inputs/IO.I107[12] <-> I107 (GSIO-A-16DIN)/Digital Inputs/Channel 12
//     Task_P1 Inputs/IO.I107[13] <-> I107 (GSIO-A-16DIN)/Digital Inputs/Channel 13
//     Task_P1 Inputs/IO.I107[14] <-> I107 (GSIO-A-16DIN)/Digital Inputs/Channel 14
//     Task_P1 Inputs/IO.I107[15] <-> I107 (GSIO-A-16DIN)/Digital Inputs/Channel 15
//     Task_P1 Inputs/IO.I107[16] <-> I107 (GSIO-A-16DIN)/Digital Inputs/Channel 16
//     Task_P1 Inputs/IO.I107[1] <-> I107 (GSIO-A-16DIN)/Digital Inputs/Channel 1
//     Task_P1 Inputs/IO.I107[2] <-> I107 (GSIO-A-16DIN)/Digital Inputs/Channel 2
//     Task_P1 Inputs/IO.I107[3] <-> I107 (GSIO-A-16DIN)/Digital Inputs/Channel 3
//     Task_P1 Inputs/IO.I107[4] <-> I107 (GSIO-A-16DIN)/Digital Inputs/Channel 4
//     Task_P1 Inputs/IO.I107[5] <-> I107 (GSIO-A-16DIN)/Digital Inputs/Channel 5
//     Task_P1 Inputs/IO.I107[6] <-> I107 (GSIO-A-16DIN)/Digital Inputs/Channel 6
//     Task_P1 Inputs/IO.I107[7] <-> I107 (GSIO-A-16DIN)/Digital Inputs/Channel 7
//     Task_P1 Inputs/IO.I107[8] <-> I107 (GSIO-A-16DIN)/Digital Inputs/Channel 8
//     Task_P1 Inputs/IO.I107[9] <-> I107 (GSIO-A-16DIN)/Digital Inputs/Channel 9
//     Task_P1 Inputs/IO.I108[10] <-> I108 (GSIO-A-16DIN)/Digital Inputs/Channel 10
//     Task_P1 Inputs/IO.I108[11] <-> I108 (GSIO-A-16DIN)/Digital Inputs/Channel 11
//     Task_P1 Inputs/IO.I108[12] <-> I108 (GSIO-A-16DIN)/Digital Inputs/Channel 12
//     Task_P1 Inputs/IO.I108[13] <-> I108 (GSIO-A-16DIN)/Digital Inputs/Channel 13
//     Task_P1 Inputs/IO.I108[14] <-> I108 (GSIO-A-16DIN)/Digital Inputs/Channel 14
//     Task_P1 Inputs/IO.I108[15] <-> I108 (GSIO-A-16DIN)/Digital Inputs/Channel 15
//     Task_P1 Inputs/IO.I108[16] <-> I108 (GSIO-A-16DIN)/Digital Inputs/Channel 16
//     Task_P1 Inputs/IO.I108[1] <-> I108 (GSIO-A-16DIN)/Digital Inputs/Channel 1
//     Task_P1 Inputs/IO.I108[2] <-> I108 (GSIO-A-16DIN)/Digital Inputs/Channel 2
//     Task_P1 Inputs/IO.I108[3] <-> I108 (GSIO-A-16DIN)/Digital Inputs/Channel 3
//     Task_P1 Inputs/IO.I108[4] <-> I108 (GSIO-A-16DIN)/Digital Inputs/Channel 4
//     Task_P1 Inputs/IO.I108[5] <-> I108 (GSIO-A-16DIN)/Digital Inputs/Channel 5
//     Task_P1 Inputs/IO.I108[6] <-> I108 (GSIO-A-16DIN)/Digital Inputs/Channel 6
//     Task_P1 Inputs/IO.I108[7] <-> I108 (GSIO-A-16DIN)/Digital Inputs/Channel 7
//     Task_P1 Inputs/IO.I108[8] <-> I108 (GSIO-A-16DIN)/Digital Inputs/Channel 8
//     Task_P1 Inputs/IO.I108[9] <-> I108 (GSIO-A-16DIN)/Digital Inputs/Channel 9
//     Task_P1 Inputs/IO.I109[10] <-> I109 (GSIO-A-16DIN)/Digital Inputs/Channel 10
//     Task_P1 Inputs/IO.I109[11] <-> I109 (GSIO-A-16DIN)/Digital Inputs/Channel 11
//     Task_P1 Inputs/IO.I109[12] <-> I109 (GSIO-A-16DIN)/Digital Inputs/Channel 12
//     Task_P1 Inputs/IO.I109[13] <-> I109 (GSIO-A-16DIN)/Digital Inputs/Channel 13
//     Task_P1 Inputs/IO.I109[14] <-> I109 (GSIO-A-16DIN)/Digital Inputs/Channel 14
//     Task_P1 Inputs/IO.I109[15] <-> I109 (GSIO-A-16DIN)/Digital Inputs/Channel 15
//     Task_P1 Inputs/IO.I109[16] <-> I109 (GSIO-A-16DIN)/Digital Inputs/Channel 16
//     Task_P1 Inputs/IO.I109[1] <-> I109 (GSIO-A-16DIN)/Digital Inputs/Channel 1
//     Task_P1 Inputs/IO.I109[2] <-> I109 (GSIO-A-16DIN)/Digital Inputs/Channel 2
//     Task_P1 Inputs/IO.I109[3] <-> I109 (GSIO-A-16DIN)/Digital Inputs/Channel 3
//     Task_P1 Inputs/IO.I109[4] <-> I109 (GSIO-A-16DIN)/Digital Inputs/Channel 4
//     Task_P1 Inputs/IO.I109[5] <-> I109 (GSIO-A-16DIN)/Digital Inputs/Channel 5
//     Task_P1 Inputs/IO.I109[6] <-> I109 (GSIO-A-16DIN)/Digital Inputs/Channel 6
//     Task_P1 Inputs/IO.I109[7] <-> I109 (GSIO-A-16DIN)/Digital Inputs/Channel 7
//     Task_P1 Inputs/IO.I109[8] <-> I109 (GSIO-A-16DIN)/Digital Inputs/Channel 8
//     Task_P1 Inputs/IO.I109[9] <-> I109 (GSIO-A-16DIN)/Digital Inputs/Channel 9
//     Task_P1 Outputs/IO.AO101[{0..3}] <-> AO101 (GSIO-A-4AOV)/Analog Outputs/Channel {1..4}  (4 links)
//     Task_P1 Outputs/IO.Q101[10] <-> Q101 (GSIO-A-16DON)/Digital Outputs/Channel 10
//     Task_P1 Outputs/IO.Q101[11] <-> Q101 (GSIO-A-16DON)/Digital Outputs/Channel 11
//     Task_P1 Outputs/IO.Q101[12] <-> Q101 (GSIO-A-16DON)/Digital Outputs/Channel 12
//     Task_P1 Outputs/IO.Q101[13] <-> Q101 (GSIO-A-16DON)/Digital Outputs/Channel 13
//     Task_P1 Outputs/IO.Q101[14] <-> Q101 (GSIO-A-16DON)/Digital Outputs/Channel 14
//     Task_P1 Outputs/IO.Q101[15] <-> Q101 (GSIO-A-16DON)/Digital Outputs/Channel 15
//     Task_P1 Outputs/IO.Q101[16] <-> Q101 (GSIO-A-16DON)/Digital Outputs/Channel 16
//     Task_P1 Outputs/IO.Q101[1] <-> Q101 (GSIO-A-16DON)/Digital Outputs/Channel 1
//     Task_P1 Outputs/IO.Q101[2] <-> Q101 (GSIO-A-16DON)/Digital Outputs/Channel 2
//     Task_P1 Outputs/IO.Q101[3] <-> Q101 (GSIO-A-16DON)/Digital Outputs/Channel 3
//     Task_P1 Outputs/IO.Q101[4] <-> Q101 (GSIO-A-16DON)/Digital Outputs/Channel 4
//     Task_P1 Outputs/IO.Q101[5] <-> Q101 (GSIO-A-16DON)/Digital Outputs/Channel 5
//     Task_P1 Outputs/IO.Q101[6] <-> Q101 (GSIO-A-16DON)/Digital Outputs/Channel 6
//     Task_P1 Outputs/IO.Q101[7] <-> Q101 (GSIO-A-16DON)/Digital Outputs/Channel 7
//     Task_P1 Outputs/IO.Q101[8] <-> Q101 (GSIO-A-16DON)/Digital Outputs/Channel 8
//     Task_P1 Outputs/IO.Q101[9] <-> Q101 (GSIO-A-16DON)/Digital Outputs/Channel 9
//     Task_P1 Outputs/IO.Q102[10] <-> Q102 (GSIO-A-16DON)/Digital Outputs/Channel 10
//     Task_P1 Outputs/IO.Q102[11] <-> Q102 (GSIO-A-16DON)/Digital Outputs/Channel 11
//     Task_P1 Outputs/IO.Q102[12] <-> Q102 (GSIO-A-16DON)/Digital Outputs/Channel 12
//     Task_P1 Outputs/IO.Q102[13] <-> Q102 (GSIO-A-16DON)/Digital Outputs/Channel 13
//     Task_P1 Outputs/IO.Q102[14] <-> Q102 (GSIO-A-16DON)/Digital Outputs/Channel 14
//     Task_P1 Outputs/IO.Q102[15] <-> Q102 (GSIO-A-16DON)/Digital Outputs/Channel 15
//     Task_P1 Outputs/IO.Q102[16] <-> Q102 (GSIO-A-16DON)/Digital Outputs/Channel 16
//     Task_P1 Outputs/IO.Q102[1] <-> Q102 (GSIO-A-16DON)/Digital Outputs/Channel 1
//     Task_P1 Outputs/IO.Q102[2] <-> Q102 (GSIO-A-16DON)/Digital Outputs/Channel 2
//     Task_P1 Outputs/IO.Q102[3] <-> Q102 (GSIO-A-16DON)/Digital Outputs/Channel 3
//     Task_P1 Outputs/IO.Q102[4] <-> Q102 (GSIO-A-16DON)/Digital Outputs/Channel 4
//     Task_P1 Outputs/IO.Q102[5] <-> Q102 (GSIO-A-16DON)/Digital Outputs/Channel 5
//     Task_P1 Outputs/IO.Q102[6] <-> Q102 (GSIO-A-16DON)/Digital Outputs/Channel 6
//     Task_P1 Outputs/IO.Q102[7] <-> Q102 (GSIO-A-16DON)/Digital Outputs/Channel 7
//     Task_P1 Outputs/IO.Q102[8] <-> Q102 (GSIO-A-16DON)/Digital Outputs/Channel 8
//     Task_P1 Outputs/IO.Q102[9] <-> Q102 (GSIO-A-16DON)/Digital Outputs/Channel 9
//     Task_P1 Outputs/IO.Q103[10] <-> Q103 (GSIO-A-16DON)/Digital Outputs/Channel 10
//     Task_P1 Outputs/IO.Q103[11] <-> Q103 (GSIO-A-16DON)/Digital Outputs/Channel 11
//     Task_P1 Outputs/IO.Q103[12] <-> Q103 (GSIO-A-16DON)/Digital Outputs/Channel 12
//     Task_P1 Outputs/IO.Q103[13] <-> Q103 (GSIO-A-16DON)/Digital Outputs/Channel 13
//     Task_P1 Outputs/IO.Q103[14] <-> Q103 (GSIO-A-16DON)/Digital Outputs/Channel 14
//     Task_P1 Outputs/IO.Q103[15] <-> Q103 (GSIO-A-16DON)/Digital Outputs/Channel 15
//     Task_P1 Outputs/IO.Q103[16] <-> Q103 (GSIO-A-16DON)/Digital Outputs/Channel 16
//     Task_P1 Outputs/IO.Q103[1] <-> Q103 (GSIO-A-16DON)/Digital Outputs/Channel 1
//     Task_P1 Outputs/IO.Q103[2] <-> Q103 (GSIO-A-16DON)/Digital Outputs/Channel 2
//     Task_P1 Outputs/IO.Q103[3] <-> Q103 (GSIO-A-16DON)/Digital Outputs/Channel 3
//     Task_P1 Outputs/IO.Q103[4] <-> Q103 (GSIO-A-16DON)/Digital Outputs/Channel 4
//     Task_P1 Outputs/IO.Q103[5] <-> Q103 (GSIO-A-16DON)/Digital Outputs/Channel 5
//     Task_P1 Outputs/IO.Q103[6] <-> Q103 (GSIO-A-16DON)/Digital Outputs/Channel 6
//     Task_P1 Outputs/IO.Q103[7] <-> Q103 (GSIO-A-16DON)/Digital Outputs/Channel 7
//     Task_P1 Outputs/IO.Q103[8] <-> Q103 (GSIO-A-16DON)/Digital Outputs/Channel 8
//     Task_P1 Outputs/IO.Q103[9] <-> Q103 (GSIO-A-16DON)/Digital Outputs/Channel 9
//     Task_P1 Outputs/IO.Q104[10] <-> Q104 (GSIO-A-16DON)/Digital Outputs/Channel 10
//     Task_P1 Outputs/IO.Q104[11] <-> Q104 (GSIO-A-16DON)/Digital Outputs/Channel 11
//     Task_P1 Outputs/IO.Q104[12] <-> Q104 (GSIO-A-16DON)/Digital Outputs/Channel 12
//     Task_P1 Outputs/IO.Q104[13] <-> Q104 (GSIO-A-16DON)/Digital Outputs/Channel 13
//     Task_P1 Outputs/IO.Q104[14] <-> Q104 (GSIO-A-16DON)/Digital Outputs/Channel 14
//     Task_P1 Outputs/IO.Q104[15] <-> Q104 (GSIO-A-16DON)/Digital Outputs/Channel 15
//     Task_P1 Outputs/IO.Q104[16] <-> Q104 (GSIO-A-16DON)/Digital Outputs/Channel 16
//     Task_P1 Outputs/IO.Q104[1] <-> Q104 (GSIO-A-16DON)/Digital Outputs/Channel 1
//     Task_P1 Outputs/IO.Q104[2] <-> Q104 (GSIO-A-16DON)/Digital Outputs/Channel 2
//     Task_P1 Outputs/IO.Q104[3] <-> Q104 (GSIO-A-16DON)/Digital Outputs/Channel 3
//     Task_P1 Outputs/IO.Q104[4] <-> Q104 (GSIO-A-16DON)/Digital Outputs/Channel 4
//     Task_P1 Outputs/IO.Q104[5] <-> Q104 (GSIO-A-16DON)/Digital Outputs/Channel 5
//     Task_P1 Outputs/IO.Q104[6] <-> Q104 (GSIO-A-16DON)/Digital Outputs/Channel 6
//     Task_P1 Outputs/IO.Q104[7] <-> Q104 (GSIO-A-16DON)/Digital Outputs/Channel 7
//     Task_P1 Outputs/IO.Q104[8] <-> Q104 (GSIO-A-16DON)/Digital Outputs/Channel 8
//     Task_P1 Outputs/IO.Q104[9] <-> Q104 (GSIO-A-16DON)/Digital Outputs/Channel 9
//     Task_P1 Outputs/IO.Q105[10] <-> Q105 (GSIO-A-16DON)/Digital Outputs/Channel 10
//     Task_P1 Outputs/IO.Q105[11] <-> Q105 (GSIO-A-16DON)/Digital Outputs/Channel 11
//     Task_P1 Outputs/IO.Q105[12] <-> Q105 (GSIO-A-16DON)/Digital Outputs/Channel 12
//     Task_P1 Outputs/IO.Q105[13] <-> Q105 (GSIO-A-16DON)/Digital Outputs/Channel 13
//     Task_P1 Outputs/IO.Q105[14] <-> Q105 (GSIO-A-16DON)/Digital Outputs/Channel 14
//     Task_P1 Outputs/IO.Q105[15] <-> Q105 (GSIO-A-16DON)/Digital Outputs/Channel 15
//     Task_P1 Outputs/IO.Q105[16] <-> Q105 (GSIO-A-16DON)/Digital Outputs/Channel 16
//     Task_P1 Outputs/IO.Q105[1] <-> Q105 (GSIO-A-16DON)/Digital Outputs/Channel 1
//     Task_P1 Outputs/IO.Q105[2] <-> Q105 (GSIO-A-16DON)/Digital Outputs/Channel 2
//     Task_P1 Outputs/IO.Q105[3] <-> Q105 (GSIO-A-16DON)/Digital Outputs/Channel 3
//     Task_P1 Outputs/IO.Q105[4] <-> Q105 (GSIO-A-16DON)/Digital Outputs/Channel 4
//     Task_P1 Outputs/IO.Q105[5] <-> Q105 (GSIO-A-16DON)/Digital Outputs/Channel 5
//     Task_P1 Outputs/IO.Q105[6] <-> Q105 (GSIO-A-16DON)/Digital Outputs/Channel 6
//     Task_P1 Outputs/IO.Q105[7] <-> Q105 (GSIO-A-16DON)/Digital Outputs/Channel 7
//     Task_P1 Outputs/IO.Q105[8] <-> Q105 (GSIO-A-16DON)/Digital Outputs/Channel 8
//     Task_P1 Outputs/IO.Q105[9] <-> Q105 (GSIO-A-16DON)/Digital Outputs/Channel 9
//     Task_P1 Outputs/IO.Q106[10] <-> Q106 (GSIO-A-16DON)/Digital Outputs/Channel 10
//     Task_P1 Outputs/IO.Q106[11] <-> Q106 (GSIO-A-16DON)/Digital Outputs/Channel 11
//     Task_P1 Outputs/IO.Q106[12] <-> Q106 (GSIO-A-16DON)/Digital Outputs/Channel 12
//     Task_P1 Outputs/IO.Q106[13] <-> Q106 (GSIO-A-16DON)/Digital Outputs/Channel 13
//     Task_P1 Outputs/IO.Q106[14] <-> Q106 (GSIO-A-16DON)/Digital Outputs/Channel 14
//     Task_P1 Outputs/IO.Q106[15] <-> Q106 (GSIO-A-16DON)/Digital Outputs/Channel 15
//     Task_P1 Outputs/IO.Q106[16] <-> Q106 (GSIO-A-16DON)/Digital Outputs/Channel 16
//     Task_P1 Outputs/IO.Q106[1] <-> Q106 (GSIO-A-16DON)/Digital Outputs/Channel 1
//     Task_P1 Outputs/IO.Q106[2] <-> Q106 (GSIO-A-16DON)/Digital Outputs/Channel 2
//     Task_P1 Outputs/IO.Q106[3] <-> Q106 (GSIO-A-16DON)/Digital Outputs/Channel 3
//     Task_P1 Outputs/IO.Q106[4] <-> Q106 (GSIO-A-16DON)/Digital Outputs/Channel 4
//     Task_P1 Outputs/IO.Q106[5] <-> Q106 (GSIO-A-16DON)/Digital Outputs/Channel 5
//     Task_P1 Outputs/IO.Q106[6] <-> Q106 (GSIO-A-16DON)/Digital Outputs/Channel 6
//     Task_P1 Outputs/IO.Q106[7] <-> Q106 (GSIO-A-16DON)/Digital Outputs/Channel 7
//     Task_P1 Outputs/IO.Q106[8] <-> Q106 (GSIO-A-16DON)/Digital Outputs/Channel 8
//     Task_P1 Outputs/IO.Q106[9] <-> Q106 (GSIO-A-16DON)/Digital Outputs/Channel 9
//     Task_P1 Outputs/IO.Q107[10] <-> Q107 (GSIO-A-16DON)/Digital Outputs/Channel 10
//     Task_P1 Outputs/IO.Q107[11] <-> Q107 (GSIO-A-16DON)/Digital Outputs/Channel 11
//     Task_P1 Outputs/IO.Q107[12] <-> Q107 (GSIO-A-16DON)/Digital Outputs/Channel 12
//     Task_P1 Outputs/IO.Q107[13] <-> Q107 (GSIO-A-16DON)/Digital Outputs/Channel 13
//     Task_P1 Outputs/IO.Q107[14] <-> Q107 (GSIO-A-16DON)/Digital Outputs/Channel 14
//     Task_P1 Outputs/IO.Q107[15] <-> Q107 (GSIO-A-16DON)/Digital Outputs/Channel 15
//     Task_P1 Outputs/IO.Q107[16] <-> Q107 (GSIO-A-16DON)/Digital Outputs/Channel 16
//     Task_P1 Outputs/IO.Q107[1] <-> Q107 (GSIO-A-16DON)/Digital Outputs/Channel 1
//     Task_P1 Outputs/IO.Q107[2] <-> Q107 (GSIO-A-16DON)/Digital Outputs/Channel 2
//     Task_P1 Outputs/IO.Q107[3] <-> Q107 (GSIO-A-16DON)/Digital Outputs/Channel 3
//     Task_P1 Outputs/IO.Q107[4] <-> Q107 (GSIO-A-16DON)/Digital Outputs/Channel 4
//     Task_P1 Outputs/IO.Q107[5] <-> Q107 (GSIO-A-16DON)/Digital Outputs/Channel 5
//     Task_P1 Outputs/IO.Q107[6] <-> Q107 (GSIO-A-16DON)/Digital Outputs/Channel 6
//     Task_P1 Outputs/IO.Q107[7] <-> Q107 (GSIO-A-16DON)/Digital Outputs/Channel 7
//     Task_P1 Outputs/IO.Q107[8] <-> Q107 (GSIO-A-16DON)/Digital Outputs/Channel 8
//     Task_P1 Outputs/IO.Q107[9] <-> Q107 (GSIO-A-16DON)/Digital Outputs/Channel 9
//     Task_P1 Outputs/IO.Q108[10] <-> Q108 (GSIO-A-16DON)/Digital Outputs/Channel 10
//     Task_P1 Outputs/IO.Q108[11] <-> Q108 (GSIO-A-16DON)/Digital Outputs/Channel 11
//     Task_P1 Outputs/IO.Q108[12] <-> Q108 (GSIO-A-16DON)/Digital Outputs/Channel 12
//     Task_P1 Outputs/IO.Q108[13] <-> Q108 (GSIO-A-16DON)/Digital Outputs/Channel 13
//     Task_P1 Outputs/IO.Q108[14] <-> Q108 (GSIO-A-16DON)/Digital Outputs/Channel 14
//     Task_P1 Outputs/IO.Q108[15] <-> Q108 (GSIO-A-16DON)/Digital Outputs/Channel 15
//     Task_P1 Outputs/IO.Q108[16] <-> Q108 (GSIO-A-16DON)/Digital Outputs/Channel 16
//     Task_P1 Outputs/IO.Q108[1] <-> Q108 (GSIO-A-16DON)/Digital Outputs/Channel 1
//     Task_P1 Outputs/IO.Q108[2] <-> Q108 (GSIO-A-16DON)/Digital Outputs/Channel 2
//     Task_P1 Outputs/IO.Q108[3] <-> Q108 (GSIO-A-16DON)/Digital Outputs/Channel 3
//     Task_P1 Outputs/IO.Q108[4] <-> Q108 (GSIO-A-16DON)/Digital Outputs/Channel 4
//     Task_P1 Outputs/IO.Q108[5] <-> Q108 (GSIO-A-16DON)/Digital Outputs/Channel 5
//     Task_P1 Outputs/IO.Q108[6] <-> Q108 (GSIO-A-16DON)/Digital Outputs/Channel 6
//     Task_P1 Outputs/IO.Q108[7] <-> Q108 (GSIO-A-16DON)/Digital Outputs/Channel 7
//     Task_P1 Outputs/IO.Q108[8] <-> Q108 (GSIO-A-16DON)/Digital Outputs/Channel 8
//     Task_P1 Outputs/IO.Q108[9] <-> Q108 (GSIO-A-16DON)/Digital Outputs/Channel 9
//     Task_P1 Outputs/IO.Q109[10] <-> Q109 (GSIO-A-16DON)/Digital Outputs/Channel 10
//     Task_P1 Outputs/IO.Q109[11] <-> Q109 (GSIO-A-16DON)/Digital Outputs/Channel 11
//     Task_P1 Outputs/IO.Q109[12] <-> Q109 (GSIO-A-16DON)/Digital Outputs/Channel 12
//     Task_P1 Outputs/IO.Q109[13] <-> Q109 (GSIO-A-16DON)/Digital Outputs/Channel 13
//     Task_P1 Outputs/IO.Q109[14] <-> Q109 (GSIO-A-16DON)/Digital Outputs/Channel 14
//     Task_P1 Outputs/IO.Q109[15] <-> Q109 (GSIO-A-16DON)/Digital Outputs/Channel 15
//     Task_P1 Outputs/IO.Q109[16] <-> Q109 (GSIO-A-16DON)/Digital Outputs/Channel 16
//     Task_P1 Outputs/IO.Q109[1] <-> Q109 (GSIO-A-16DON)/Digital Outputs/Channel 1
//     Task_P1 Outputs/IO.Q109[2] <-> Q109 (GSIO-A-16DON)/Digital Outputs/Channel 2
//     Task_P1 Outputs/IO.Q109[3] <-> Q109 (GSIO-A-16DON)/Digital Outputs/Channel 3
//     Task_P1 Outputs/IO.Q109[4] <-> Q109 (GSIO-A-16DON)/Digital Outputs/Channel 4
//     Task_P1 Outputs/IO.Q109[5] <-> Q109 (GSIO-A-16DON)/Digital Outputs/Channel 5
//     Task_P1 Outputs/IO.Q109[6] <-> Q109 (GSIO-A-16DON)/Digital Outputs/Channel 6
//     Task_P1 Outputs/IO.Q109[7] <-> Q109 (GSIO-A-16DON)/Digital Outputs/Channel 7
//     Task_P1 Outputs/IO.Q109[8] <-> Q109 (GSIO-A-16DON)/Digital Outputs/Channel 8
//     Task_P1 Outputs/IO.Q109[9] <-> Q109 (GSIO-A-16DON)/Digital Outputs/Channel 9
//   MQPLC/MQPLC Instance <-> Device 3 (EtherCAT)/Box 2 (CU1128)/正极上表面除尘皮带(InoSV660N)
//     Task_P1 Inputs/GMotion.DrivesOP[18] <-> InfoData/State
//     Task_P1 Inputs/GMotion.arrAxisCtrl[18].Io.DigitalInputs <-> Inputs/Digital inputs
//     Task_P1 Inputs/GMotion.arrAxisCtrl[18].Io.ErrorCode <-> Inputs/Error code
//     Task_P1 Inputs/GMotion.iActTorque_M[18] <-> Inputs/Torque actual value
//   MQPLC/MQPLC Instance <-> Device 3 (EtherCAT)/Box 2 (CU1128)/正极下表面除尘倒装皮带(InoSV660N)
//     Task_P1 Inputs/GMotion.DrivesOP[19] <-> InfoData/State
//     Task_P1 Inputs/GMotion.arrAxisCtrl[19].Io.DigitalInputs <-> Inputs/Digital inputs
//     Task_P1 Inputs/GMotion.arrAxisCtrl[19].Io.ErrorCode <-> Inputs/Error code
//     Task_P1 Inputs/GMotion.iActTorque_M[19] <-> Inputs/Torque actual value
//   MQPLC/MQPLC Instance <-> Device 3 (EtherCAT)/Box 2 (CU1128)/正极倒角模具(InoSV660N)
//     Task_P1 Inputs/GMotion.DrivesOP[6] <-> InfoData/State
//     Task_P1 Inputs/GMotion.arrAxisCtrl[6].Io.DigitalInputs <-> Inputs/Digital inputs
//     Task_P1 Inputs/GMotion.arrAxisCtrl[6].Io.ErrorCode <-> Inputs/Error code
//     Task_P1 Inputs/GMotion.iActTorque_M[6] <-> Inputs/Torque actual value
//   MQPLC/MQPLC Instance <-> Device 3 (EtherCAT)/Box 2 (CU1128)/正极右放卷电机(InoSV660N)
//     Task_P1 Inputs/GMotion.DrivesOP[2] <-> InfoData/State
//     Task_P1 Inputs/GMotion.arrAxisCtrl[2].Io.DigitalInputs <-> Inputs/Digital inputs
//     Task_P1 Inputs/GMotion.arrAxisCtrl[2].Io.ErrorCode <-> Inputs/Error code
//     Task_P1 Inputs/GMotion.iActTorque_M[2] <-> Inputs/Torque actual value
//   MQPLC/MQPLC Instance <-> Device 3 (EtherCAT)/Box 2 (CU1128)/正极尺寸CCD压片升降(InoSV660N)
//     Task_P1 Inputs/GMotion.DrivesOP[14] <-> InfoData/State
//     Task_P1 Inputs/GMotion.arrAxisCtrl[14].Io.DigitalInputs <-> Inputs/Digital inputs
//     Task_P1 Inputs/GMotion.arrAxisCtrl[14].Io.ErrorCode <-> Inputs/Error code
//     Task_P1 Inputs/GMotion.iActTorque_M[14] <-> Inputs/Torque actual value
//   MQPLC/MQPLC Instance <-> Device 3 (EtherCAT)/Box 2 (CU1128)/正极左放卷电机(InoSV660N)
//     Task_P1 Inputs/GMotion.DrivesOP[1] <-> InfoData/State
//     Task_P1 Inputs/GMotion.arrAxisCtrl[1].Io.DigitalInputs <-> Inputs/Digital inputs
//     Task_P1 Inputs/GMotion.arrAxisCtrl[1].Io.ErrorCode <-> Inputs/Error code
//     Task_P1 Inputs/GMotion.iActTorque_M[1] <-> Inputs/Torque actual value
//   MQPLC/MQPLC Instance <-> Device 3 (EtherCAT)/Box 2 (CU1128)/正极模具纠偏X轴(肩宽)(InoSV660N)
//     Task_P1 Inputs/GMotion.DrivesOP[7] <-> InfoData/State
//     Task_P1 Inputs/GMotion.arrAxisCtrl[7].Io.DigitalInputs <-> Inputs/Digital inputs
//     Task_P1 Inputs/GMotion.arrAxisCtrl[7].Io.ErrorCode <-> Inputs/Error code
//     Task_P1 Inputs/GMotion.iActTorque_M[7] <-> Inputs/Torque actual value
//   MQPLC/MQPLC Instance <-> Device 3 (EtherCAT)/Box 2 (CU1128)/正极模具纠偏Y轴(InoSV660N)
//     Task_P1 Inputs/GMotion.DrivesOP[8] <-> InfoData/State
//     Task_P1 Inputs/GMotion.arrAxisCtrl[8].Io.DigitalInputs <-> Inputs/Digital inputs
//     Task_P1 Inputs/GMotion.arrAxisCtrl[8].Io.ErrorCode <-> Inputs/Error code
//     Task_P1 Inputs/GMotion.iActTorque_M[8] <-> Inputs/Torque actual value
//   MQPLC/MQPLC Instance <-> Device 3 (EtherCAT)/Box 2 (CU1128)/正极模切主驱动(CDHD)
//     Task_P1 Inputs/GMotion.DrivesOP[9] <-> InfoData/State
//     Task_P1 Inputs/GMotion.arrAxisCtrl[9].Io.DigitalInputs <-> TxPDO 4/Digital inputs
//     Task_P1 Inputs/GMotion.iActTorque_M[9] <-> TxPDO 1/Torque Actual Value
//   MQPLC/MQPLC Instance <-> Device 3 (EtherCAT)/Box 2 (CU1128)/正极模切前摆杆张力(InoSV660N)
//     Task_P1 Inputs/GMotion.DrivesOP[3] <-> InfoData/State
//     Task_P1 Inputs/GMotion.arrAxisCtrl[3].Io.DigitalInputs <-> Inputs/Digital inputs
//     Task_P1 Inputs/GMotion.arrAxisCtrl[3].Io.ErrorCode <-> Inputs/Error code
//     Task_P1 Inputs/GMotion.iActDriveTorque[1] <-> Inputs/Torque actual value
//     Task_P1 Outputs/GMotion.iMaxProfileVelo[1] <-> Outputs/Max profile velocity
//     Task_P1 Outputs/GMotion.iNegtiveTorqueLimits[1] <-> Outputs/Negative torque limit value
//     Task_P1 Outputs/GMotion.iPostiveTorqueLimits[1] <-> Outputs/Positive torque limit value
//     Task_P1 Outputs/GMotion.iSetDriveMode[1] <-> Outputs/Modes of operation
//     Task_P1 Outputs/GMotion.iTargetTorque[1] <-> Outputs/Target torque
//   MQPLC/MQPLC Instance <-> Device 3 (EtherCAT)/Box 2 (CU1128)/正极模切极片缓存(CDHD)
//     Task_P1 Inputs/GMotion.DrivesOP[5] <-> InfoData/State
//     Task_P1 Inputs/GMotion.arrAxisCtrl[5].Io.DigitalInputs <-> TxPDO 4/Digital inputs
//     Task_P1 Inputs/GMotion.iActTorque_M[5] <-> TxPDO 1/Torque Actual Value
//   MQPLC/MQPLC Instance <-> Device 3 (EtherCAT)/Box 2 (CU1128)/正极模切辅助驱动(InoSV660N)
//     Task_P1 Inputs/GMotion.DrivesOP[4] <-> InfoData/State
//     Task_P1 Inputs/GMotion.arrAxisCtrl[4].Io.DigitalInputs <-> Inputs/Digital inputs
//     Task_P1 Inputs/GMotion.arrAxisCtrl[4].Io.ErrorCode <-> Inputs/Error code
//     Task_P1 Inputs/GMotion.iActTorque_M[4] <-> Inputs/Torque actual value
//   MQPLC/MQPLC Instance <-> Device 3 (EtherCAT)/Box 2 (CU1128)/正极裁切切刀(InoSV660N)
//     Task_P1 Inputs/GMotion.DrivesOP[10] <-> InfoData/State
//     Task_P1 Inputs/GMotion.arrAxisCtrl[10].Io.DigitalInputs <-> Inputs/Digital inputs
//     Task_P1 Inputs/GMotion.arrAxisCtrl[10].Io.ErrorCode <-> Inputs/Error code
//     Task_P1 Inputs/GMotion.iActTorque_M[10] <-> Inputs/Torque actual value
//   MQPLC/MQPLC Instance <-> Device 3 (EtherCAT)/Box 2 (CU1128)/正极裁切角度纠偏(InoSV660N)
//     Task_P1 Inputs/GMotion.DrivesOP[11] <-> InfoData/State
//     Task_P1 Inputs/GMotion.arrAxisCtrl[11].Io.DigitalInputs <-> Inputs/Digital inputs
//     Task_P1 Inputs/GMotion.arrAxisCtrl[11].Io.ErrorCode <-> Inputs/Error code
//     Task_P1 Inputs/GMotion.iActTorque_M[11] <-> Inputs/Torque actual value
//   MQPLC/MQPLC Instance <-> Device 3 (EtherCAT)/Box 2 (CU1128)/正极裁切输送带换型(InoSV660N)
//     Task_P1 Inputs/GMotion.DrivesOP[13] <-> InfoData/State
//     Task_P1 Inputs/GMotion.arrAxisCtrl[13].Io.DigitalInputs <-> Inputs/Digital inputs
//     Task_P1 Inputs/GMotion.arrAxisCtrl[13].Io.ErrorCode <-> Inputs/Error code
//     Task_P1 Inputs/GMotion.iActTorque_M[13] <-> Inputs/Torque actual value
//   MQPLC/MQPLC Instance <-> Device 3 (EtherCAT)/Box 2 (CU1128)/正极裁切输送皮带(InoSV660N)
//     Task_P1 Inputs/GMotion.DrivesOP[12] <-> InfoData/State
//     Task_P1 Inputs/GMotion.arrAxisCtrl[12].Io.DigitalInputs <-> Inputs/Digital inputs
//     Task_P1 Inputs/GMotion.arrAxisCtrl[12].Io.ErrorCode <-> Inputs/Error code
//     Task_P1 Inputs/GMotion.iActTorque_M[12] <-> Inputs/Torque actual value
//   MQPLC/MQPLC Instance <-> Device 3 (EtherCAT)/Box 2 (CU1128)/正极踢单张废料(InoSV660N)
//     Task_P1 Inputs/GMotion.DrivesOP[17] <-> InfoData/State
//     Task_P1 Inputs/GMotion.arrAxisCtrl[17].Io.DigitalInputs <-> Inputs/Digital inputs
//     Task_P1 Inputs/GMotion.arrAxisCtrl[17].Io.ErrorCode <-> Inputs/Error code
//     Task_P1 Inputs/GMotion.iActTorque_M[17] <-> Inputs/Torque actual value
//   MQPLC/MQPLC Instance <-> Device 3 (EtherCAT)/Box 2 (CU1128)/正极踢废倒装皮带(InoSV660N)
//     Task_P1 Inputs/GMotion.DrivesOP[15] <-> InfoData/State
//     Task_P1 Inputs/GMotion.arrAxisCtrl[15].Io.DigitalInputs <-> Inputs/Digital inputs
//     Task_P1 Inputs/GMotion.arrAxisCtrl[15].Io.ErrorCode <-> Inputs/Error code
//     Task_P1 Inputs/GMotion.iActTorque_M[15] <-> Inputs/Torque actual value
//   MQPLC/MQPLC Instance <-> Device 3 (EtherCAT)/Box 2 (CU1128)/正极踢连续废料(InoSV660N)
//     Task_P1 Inputs/GMotion.DrivesOP[16] <-> InfoData/State
//     Task_P1 Inputs/GMotion.arrAxisCtrl[16].Io.DigitalInputs <-> Inputs/Digital inputs
//     Task_P1 Inputs/GMotion.arrAxisCtrl[16].Io.ErrorCode <-> Inputs/Error code
//     Task_P1 Inputs/GMotion.iActTorque_M[16] <-> Inputs/Torque actual value
//   MQPLC/MQPLC Instance <-> Device 3 (EtherCAT)/Box 2 (CU1128)/负极IO耦合器(GSIO-A-ECC)
//     Task_P1 Inputs/IO.AI201[0] <-> AI201 (GSIO-A-4AIHV)/Analog Inputs/Channel 1
//     Task_P1 Inputs/IO.AI201[1] <-> AI201 (GSIO-A-4AIHV)/Analog Inputs/Channel 2
//     Task_P1 Inputs/IO.AI201[2] <-> AI201 (GSIO-A-4AIHV)/Analog Inputs/Channel 3
//     Task_P1 Inputs/IO.AI201[3] <-> AI201 (GSIO-A-4AIHV)/Analog Inputs/Channel 4
//     Task_P1 Inputs/IO.AI202[0] <-> AI202 (GSIO-A-4AIHV)/Analog Inputs/Channel 1
//     Task_P1 Inputs/IO.AI202[1] <-> AI202 (GSIO-A-4AIHV)/Analog Inputs/Channel 2
//     Task_P1 Inputs/IO.AI202[2] <-> AI202 (GSIO-A-4AIHV)/Analog Inputs/Channel 3
//     Task_P1 Inputs/IO.AI202[3] <-> AI202 (GSIO-A-4AIHV)/Analog Inputs/Channel 4
//     Task_P1 Inputs/IO.I201[10] <-> I201 (GSIO-A-16DIN)/Digital Inputs/Channel 10
//     Task_P1 Inputs/IO.I201[11] <-> I201 (GSIO-A-16DIN)/Digital Inputs/Channel 11
//     Task_P1 Inputs/IO.I201[12] <-> I201 (GSIO-A-16DIN)/Digital Inputs/Channel 12
//     Task_P1 Inputs/IO.I201[13] <-> I201 (GSIO-A-16DIN)/Digital Inputs/Channel 13
//     Task_P1 Inputs/IO.I201[14] <-> I201 (GSIO-A-16DIN)/Digital Inputs/Channel 14
//     Task_P1 Inputs/IO.I201[15] <-> I201 (GSIO-A-16DIN)/Digital Inputs/Channel 15
//     Task_P1 Inputs/IO.I201[16] <-> I201 (GSIO-A-16DIN)/Digital Inputs/Channel 16
//     Task_P1 Inputs/IO.I201[1] <-> I201 (GSIO-A-16DIN)/Digital Inputs/Channel 1
//     Task_P1 Inputs/IO.I201[2] <-> I201 (GSIO-A-16DIN)/Digital Inputs/Channel 2
//     Task_P1 Inputs/IO.I201[3] <-> I201 (GSIO-A-16DIN)/Digital Inputs/Channel 3
//     Task_P1 Inputs/IO.I201[4] <-> I201 (GSIO-A-16DIN)/Digital Inputs/Channel 4
//     Task_P1 Inputs/IO.I201[5] <-> I201 (GSIO-A-16DIN)/Digital Inputs/Channel 5
//     Task_P1 Inputs/IO.I201[6] <-> I201 (GSIO-A-16DIN)/Digital Inputs/Channel 6
//     Task_P1 Inputs/IO.I201[7] <-> I201 (GSIO-A-16DIN)/Digital Inputs/Channel 7
//     Task_P1 Inputs/IO.I201[8] <-> I201 (GSIO-A-16DIN)/Digital Inputs/Channel 8
//     Task_P1 Inputs/IO.I201[9] <-> I201 (GSIO-A-16DIN)/Digital Inputs/Channel 9
//     Task_P1 Inputs/IO.I202[10] <-> I202 (GSIO-A-16DIN)/Digital Inputs/Channel 10
//     Task_P1 Inputs/IO.I202[11] <-> I202 (GSIO-A-16DIN)/Digital Inputs/Channel 11
//     Task_P1 Inputs/IO.I202[12] <-> I202 (GSIO-A-16DIN)/Digital Inputs/Channel 12
//     Task_P1 Inputs/IO.I202[13] <-> I202 (GSIO-A-16DIN)/Digital Inputs/Channel 13
//     Task_P1 Inputs/IO.I202[14] <-> I202 (GSIO-A-16DIN)/Digital Inputs/Channel 14
//     Task_P1 Inputs/IO.I202[15] <-> I202 (GSIO-A-16DIN)/Digital Inputs/Channel 15
//     Task_P1 Inputs/IO.I202[16] <-> I202 (GSIO-A-16DIN)/Digital Inputs/Channel 16
//     Task_P1 Inputs/IO.I202[1] <-> I202 (GSIO-A-16DIN)/Digital Inputs/Channel 1
//     Task_P1 Inputs/IO.I202[2] <-> I202 (GSIO-A-16DIN)/Digital Inputs/Channel 2
//     Task_P1 Inputs/IO.I202[3] <-> I202 (GSIO-A-16DIN)/Digital Inputs/Channel 3
//     Task_P1 Inputs/IO.I202[4] <-> I202 (GSIO-A-16DIN)/Digital Inputs/Channel 4
//     Task_P1 Inputs/IO.I202[5] <-> I202 (GSIO-A-16DIN)/Digital Inputs/Channel 5
//     Task_P1 Inputs/IO.I202[6] <-> I202 (GSIO-A-16DIN)/Digital Inputs/Channel 6
//     Task_P1 Inputs/IO.I202[7] <-> I202 (GSIO-A-16DIN)/Digital Inputs/Channel 7
//     Task_P1 Inputs/IO.I202[8] <-> I202 (GSIO-A-16DIN)/Digital Inputs/Channel 8
//     Task_P1 Inputs/IO.I202[9] <-> I202 (GSIO-A-16DIN)/Digital Inputs/Channel 9
//     Task_P1 Inputs/IO.I203[10] <-> I203 (GSIO-A-16DIN)/Digital Inputs/Channel 10
//     Task_P1 Inputs/IO.I203[11] <-> I203 (GSIO-A-16DIN)/Digital Inputs/Channel 11
//     Task_P1 Inputs/IO.I203[12] <-> I203 (GSIO-A-16DIN)/Digital Inputs/Channel 12
//     Task_P1 Inputs/IO.I203[13] <-> I203 (GSIO-A-16DIN)/Digital Inputs/Channel 13
//     Task_P1 Inputs/IO.I203[14] <-> I203 (GSIO-A-16DIN)/Digital Inputs/Channel 14
//     Task_P1 Inputs/IO.I203[15] <-> I203 (GSIO-A-16DIN)/Digital Inputs/Channel 15
//     Task_P1 Inputs/IO.I203[16] <-> I203 (GSIO-A-16DIN)/Digital Inputs/Channel 16
//     Task_P1 Inputs/IO.I203[1] <-> I203 (GSIO-A-16DIN)/Digital Inputs/Channel 1
//     Task_P1 Inputs/IO.I203[2] <-> I203 (GSIO-A-16DIN)/Digital Inputs/Channel 2
//     Task_P1 Inputs/IO.I203[3] <-> I203 (GSIO-A-16DIN)/Digital Inputs/Channel 3
//     Task_P1 Inputs/IO.I203[4] <-> I203 (GSIO-A-16DIN)/Digital Inputs/Channel 4
//     Task_P1 Inputs/IO.I203[5] <-> I203 (GSIO-A-16DIN)/Digital Inputs/Channel 5
//     Task_P1 Inputs/IO.I203[6] <-> I203 (GSIO-A-16DIN)/Digital Inputs/Channel 6
//     Task_P1 Inputs/IO.I203[7] <-> I203 (GSIO-A-16DIN)/Digital Inputs/Channel 7
//     Task_P1 Inputs/IO.I203[8] <-> I203 (GSIO-A-16DIN)/Digital Inputs/Channel 8
//     Task_P1 Inputs/IO.I203[9] <-> I203 (GSIO-A-16DIN)/Digital Inputs/Channel 9
//     Task_P1 Inputs/IO.I204[10] <-> I204 (GSIO-A-16DIN)/Digital Inputs/Channel 10
//     Task_P1 Inputs/IO.I204[11] <-> I204 (GSIO-A-16DIN)/Digital Inputs/Channel 11
//     Task_P1 Inputs/IO.I204[12] <-> I204 (GSIO-A-16DIN)/Digital Inputs/Channel 12
//     Task_P1 Inputs/IO.I204[13] <-> I204 (GSIO-A-16DIN)/Digital Inputs/Channel 13
//     Task_P1 Inputs/IO.I204[14] <-> I204 (GSIO-A-16DIN)/Digital Inputs/Channel 14
//     Task_P1 Inputs/IO.I204[15] <-> I204 (GSIO-A-16DIN)/Digital Inputs/Channel 15
//     Task_P1 Inputs/IO.I204[16] <-> I204 (GSIO-A-16DIN)/Digital Inputs/Channel 16
//     Task_P1 Inputs/IO.I204[1] <-> I204 (GSIO-A-16DIN)/Digital Inputs/Channel 1
//     Task_P1 Inputs/IO.I204[2] <-> I204 (GSIO-A-16DIN)/Digital Inputs/Channel 2
//     Task_P1 Inputs/IO.I204[3] <-> I204 (GSIO-A-16DIN)/Digital Inputs/Channel 3
//     Task_P1 Inputs/IO.I204[4] <-> I204 (GSIO-A-16DIN)/Digital Inputs/Channel 4
//     Task_P1 Inputs/IO.I204[5] <-> I204 (GSIO-A-16DIN)/Digital Inputs/Channel 5
//     Task_P1 Inputs/IO.I204[6] <-> I204 (GSIO-A-16DIN)/Digital Inputs/Channel 6
//     Task_P1 Inputs/IO.I204[7] <-> I204 (GSIO-A-16DIN)/Digital Inputs/Channel 7
//     Task_P1 Inputs/IO.I204[8] <-> I204 (GSIO-A-16DIN)/Digital Inputs/Channel 8
//     Task_P1 Inputs/IO.I204[9] <-> I204 (GSIO-A-16DIN)/Digital Inputs/Channel 9
//     Task_P1 Inputs/IO.I205[10] <-> I205 (GSIO-A-16DIN)/Digital Inputs/Channel 10
//     Task_P1 Inputs/IO.I205[11] <-> I205 (GSIO-A-16DIN)/Digital Inputs/Channel 11
//     Task_P1 Inputs/IO.I205[12] <-> I205 (GSIO-A-16DIN)/Digital Inputs/Channel 12
//     Task_P1 Inputs/IO.I205[13] <-> I205 (GSIO-A-16DIN)/Digital Inputs/Channel 13
//     Task_P1 Inputs/IO.I205[14] <-> I205 (GSIO-A-16DIN)/Digital Inputs/Channel 14
//     Task_P1 Inputs/IO.I205[15] <-> I205 (GSIO-A-16DIN)/Digital Inputs/Channel 15
//     Task_P1 Inputs/IO.I205[16] <-> I205 (GSIO-A-16DIN)/Digital Inputs/Channel 16
//     Task_P1 Inputs/IO.I205[1] <-> I205 (GSIO-A-16DIN)/Digital Inputs/Channel 1
//     Task_P1 Inputs/IO.I205[2] <-> I205 (GSIO-A-16DIN)/Digital Inputs/Channel 2
//     Task_P1 Inputs/IO.I205[3] <-> I205 (GSIO-A-16DIN)/Digital Inputs/Channel 3
//     Task_P1 Inputs/IO.I205[4] <-> I205 (GSIO-A-16DIN)/Digital Inputs/Channel 4
//     Task_P1 Inputs/IO.I205[5] <-> I205 (GSIO-A-16DIN)/Digital Inputs/Channel 5
//     Task_P1 Inputs/IO.I205[6] <-> I205 (GSIO-A-16DIN)/Digital Inputs/Channel 6
//     Task_P1 Inputs/IO.I205[7] <-> I205 (GSIO-A-16DIN)/Digital Inputs/Channel 7
//     Task_P1 Inputs/IO.I205[8] <-> I205 (GSIO-A-16DIN)/Digital Inputs/Channel 8
//     Task_P1 Inputs/IO.I205[9] <-> I205 (GSIO-A-16DIN)/Digital Inputs/Channel 9
//     Task_P1 Inputs/IO.I206[10] <-> I206 (GSIO-A-16DIN)/Digital Inputs/Channel 10
//     Task_P1 Inputs/IO.I206[11] <-> I206 (GSIO-A-16DIN)/Digital Inputs/Channel 11
//     Task_P1 Inputs/IO.I206[12] <-> I206 (GSIO-A-16DIN)/Digital Inputs/Channel 12
//     Task_P1 Inputs/IO.I206[13] <-> I206 (GSIO-A-16DIN)/Digital Inputs/Channel 13
//     Task_P1 Inputs/IO.I206[14] <-> I206 (GSIO-A-16DIN)/Digital Inputs/Channel 14
//     Task_P1 Inputs/IO.I206[15] <-> I206 (GSIO-A-16DIN)/Digital Inputs/Channel 15
//     Task_P1 Inputs/IO.I206[16] <-> I206 (GSIO-A-16DIN)/Digital Inputs/Channel 16
//     Task_P1 Inputs/IO.I206[1] <-> I206 (GSIO-A-16DIN)/Digital Inputs/Channel 1
//     Task_P1 Inputs/IO.I206[2] <-> I206 (GSIO-A-16DIN)/Digital Inputs/Channel 2
//     Task_P1 Inputs/IO.I206[3] <-> I206 (GSIO-A-16DIN)/Digital Inputs/Channel 3
//     Task_P1 Inputs/IO.I206[4] <-> I206 (GSIO-A-16DIN)/Digital Inputs/Channel 4
//     Task_P1 Inputs/IO.I206[5] <-> I206 (GSIO-A-16DIN)/Digital Inputs/Channel 5
//     Task_P1 Inputs/IO.I206[6] <-> I206 (GSIO-A-16DIN)/Digital Inputs/Channel 6
//     Task_P1 Inputs/IO.I206[7] <-> I206 (GSIO-A-16DIN)/Digital Inputs/Channel 7
//     Task_P1 Inputs/IO.I206[8] <-> I206 (GSIO-A-16DIN)/Digital Inputs/Channel 8
//     Task_P1 Inputs/IO.I206[9] <-> I206 (GSIO-A-16DIN)/Digital Inputs/Channel 9
//     Task_P1 Inputs/IO.I207[10] <-> I207 (GSIO-A-16DIN)/Digital Inputs/Channel 10
//     Task_P1 Inputs/IO.I207[11] <-> I207 (GSIO-A-16DIN)/Digital Inputs/Channel 11
//     Task_P1 Inputs/IO.I207[12] <-> I207 (GSIO-A-16DIN)/Digital Inputs/Channel 12
//     Task_P1 Inputs/IO.I207[13] <-> I207 (GSIO-A-16DIN)/Digital Inputs/Channel 13
//     Task_P1 Inputs/IO.I207[14] <-> I207 (GSIO-A-16DIN)/Digital Inputs/Channel 14
//     Task_P1 Inputs/IO.I207[15] <-> I207 (GSIO-A-16DIN)/Digital Inputs/Channel 15
//     Task_P1 Inputs/IO.I207[16] <-> I207 (GSIO-A-16DIN)/Digital Inputs/Channel 16
//     Task_P1 Inputs/IO.I207[1] <-> I207 (GSIO-A-16DIN)/Digital Inputs/Channel 1
//     Task_P1 Inputs/IO.I207[2] <-> I207 (GSIO-A-16DIN)/Digital Inputs/Channel 2
//     Task_P1 Inputs/IO.I207[3] <-> I207 (GSIO-A-16DIN)/Digital Inputs/Channel 3
//     Task_P1 Inputs/IO.I207[4] <-> I207 (GSIO-A-16DIN)/Digital Inputs/Channel 4
//     Task_P1 Inputs/IO.I207[5] <-> I207 (GSIO-A-16DIN)/Digital Inputs/Channel 5
//     Task_P1 Inputs/IO.I207[6] <-> I207 (GSIO-A-16DIN)/Digital Inputs/Channel 6
//     Task_P1 Inputs/IO.I207[7] <-> I207 (GSIO-A-16DIN)/Digital Inputs/Channel 7
//     Task_P1 Inputs/IO.I207[8] <-> I207 (GSIO-A-16DIN)/Digital Inputs/Channel 8
//     Task_P1 Inputs/IO.I207[9] <-> I207 (GSIO-A-16DIN)/Digital Inputs/Channel 9
//     Task_P1 Inputs/IO.I208[10] <-> I208 (GSIO-A-16DIN)/Digital Inputs/Channel 10
//     Task_P1 Inputs/IO.I208[11] <-> I208 (GSIO-A-16DIN)/Digital Inputs/Channel 11
//     Task_P1 Inputs/IO.I208[12] <-> I208 (GSIO-A-16DIN)/Digital Inputs/Channel 12
//     Task_P1 Inputs/IO.I208[13] <-> I208 (GSIO-A-16DIN)/Digital Inputs/Channel 13
//     Task_P1 Inputs/IO.I208[14] <-> I208 (GSIO-A-16DIN)/Digital Inputs/Channel 14
//     Task_P1 Inputs/IO.I208[15] <-> I208 (GSIO-A-16DIN)/Digital Inputs/Channel 15
//     Task_P1 Inputs/IO.I208[16] <-> I208 (GSIO-A-16DIN)/Digital Inputs/Channel 16
//     Task_P1 Inputs/IO.I208[1] <-> I208 (GSIO-A-16DIN)/Digital Inputs/Channel 1
//     Task_P1 Inputs/IO.I208[2] <-> I208 (GSIO-A-16DIN)/Digital Inputs/Channel 2
//     Task_P1 Inputs/IO.I208[3] <-> I208 (GSIO-A-16DIN)/Digital Inputs/Channel 3
//     Task_P1 Inputs/IO.I208[4] <-> I208 (GSIO-A-16DIN)/Digital Inputs/Channel 4
//     Task_P1 Inputs/IO.I208[5] <-> I208 (GSIO-A-16DIN)/Digital Inputs/Channel 5
//     Task_P1 Inputs/IO.I208[6] <-> I208 (GSIO-A-16DIN)/Digital Inputs/Channel 6
//     Task_P1 Inputs/IO.I208[7] <-> I208 (GSIO-A-16DIN)/Digital Inputs/Channel 7
//     Task_P1 Inputs/IO.I208[8] <-> I208 (GSIO-A-16DIN)/Digital Inputs/Channel 8
//     Task_P1 Inputs/IO.I208[9] <-> I208 (GSIO-A-16DIN)/Digital Inputs/Channel 9
//     Task_P1 Inputs/IO.I209[10] <-> I209 (GSIO-A-16DIN)/Digital Inputs/Channel 10
//     Task_P1 Inputs/IO.I209[11] <-> I209 (GSIO-A-16DIN)/Digital Inputs/Channel 11
//     Task_P1 Inputs/IO.I209[12] <-> I209 (GSIO-A-16DIN)/Digital Inputs/Channel 12
//     Task_P1 Inputs/IO.I209[13] <-> I209 (GSIO-A-16DIN)/Digital Inputs/Channel 13
//     Task_P1 Inputs/IO.I209[14] <-> I209 (GSIO-A-16DIN)/Digital Inputs/Channel 14
//     Task_P1 Inputs/IO.I209[15] <-> I209 (GSIO-A-16DIN)/Digital Inputs/Channel 15
//     Task_P1 Inputs/IO.I209[16] <-> I209 (GSIO-A-16DIN)/Digital Inputs/Channel 16
//     Task_P1 Inputs/IO.I209[1] <-> I209 (GSIO-A-16DIN)/Digital Inputs/Channel 1
//     Task_P1 Inputs/IO.I209[2] <-> I209 (GSIO-A-16DIN)/Digital Inputs/Channel 2
//     Task_P1 Inputs/IO.I209[3] <-> I209 (GSIO-A-16DIN)/Digital Inputs/Channel 3
//     Task_P1 Inputs/IO.I209[4] <-> I209 (GSIO-A-16DIN)/Digital Inputs/Channel 4
//     Task_P1 Inputs/IO.I209[5] <-> I209 (GSIO-A-16DIN)/Digital Inputs/Channel 5
//     Task_P1 Inputs/IO.I209[6] <-> I209 (GSIO-A-16DIN)/Digital Inputs/Channel 6
//     Task_P1 Inputs/IO.I209[7] <-> I209 (GSIO-A-16DIN)/Digital Inputs/Channel 7
//     Task_P1 Inputs/IO.I209[8] <-> I209 (GSIO-A-16DIN)/Digital Inputs/Channel 8
//     Task_P1 Inputs/IO.I209[9] <-> I209 (GSIO-A-16DIN)/Digital Inputs/Channel 9
//     Task_P1 Outputs/IO.AO201[{0..3}] <-> AO201 (GSIO-A-4AOV)/Analog Outputs/Channel {1..4}  (4 links)
//     Task_P1 Outputs/IO.Q201[10] <-> Q201 (GSIO-A-16DON)/Digital Outputs/Channel 10
//     Task_P1 Outputs/IO.Q201[11] <-> Q201 (GSIO-A-16DON)/Digital Outputs/Channel 11
//     Task_P1 Outputs/IO.Q201[12] <-> Q201 (GSIO-A-16DON)/Digital Outputs/Channel 12
//     Task_P1 Outputs/IO.Q201[13] <-> Q201 (GSIO-A-16DON)/Digital Outputs/Channel 13
//     Task_P1 Outputs/IO.Q201[14] <-> Q201 (GSIO-A-16DON)/Digital Outputs/Channel 14
//     Task_P1 Outputs/IO.Q201[15] <-> Q201 (GSIO-A-16DON)/Digital Outputs/Channel 15
//     Task_P1 Outputs/IO.Q201[16] <-> Q201 (GSIO-A-16DON)/Digital Outputs/Channel 16
//     Task_P1 Outputs/IO.Q201[1] <-> Q201 (GSIO-A-16DON)/Digital Outputs/Channel 1
//     Task_P1 Outputs/IO.Q201[2] <-> Q201 (GSIO-A-16DON)/Digital Outputs/Channel 2
//     Task_P1 Outputs/IO.Q201[3] <-> Q201 (GSIO-A-16DON)/Digital Outputs/Channel 3
//     Task_P1 Outputs/IO.Q201[4] <-> Q201 (GSIO-A-16DON)/Digital Outputs/Channel 4
//     Task_P1 Outputs/IO.Q201[5] <-> Q201 (GSIO-A-16DON)/Digital Outputs/Channel 5
//     Task_P1 Outputs/IO.Q201[6] <-> Q201 (GSIO-A-16DON)/Digital Outputs/Channel 6
//     Task_P1 Outputs/IO.Q201[7] <-> Q201 (GSIO-A-16DON)/Digital Outputs/Channel 7
//     Task_P1 Outputs/IO.Q201[8] <-> Q201 (GSIO-A-16DON)/Digital Outputs/Channel 8
//     Task_P1 Outputs/IO.Q201[9] <-> Q201 (GSIO-A-16DON)/Digital Outputs/Channel 9
//     Task_P1 Outputs/IO.Q202[10] <-> Q202 (GSIO-A-16DON)/Digital Outputs/Channel 10
//     Task_P1 Outputs/IO.Q202[11] <-> Q202 (GSIO-A-16DON)/Digital Outputs/Channel 11
//     Task_P1 Outputs/IO.Q202[12] <-> Q202 (GSIO-A-16DON)/Digital Outputs/Channel 12
//     Task_P1 Outputs/IO.Q202[13] <-> Q202 (GSIO-A-16DON)/Digital Outputs/Channel 13
//     Task_P1 Outputs/IO.Q202[14] <-> Q202 (GSIO-A-16DON)/Digital Outputs/Channel 14
//     Task_P1 Outputs/IO.Q202[15] <-> Q202 (GSIO-A-16DON)/Digital Outputs/Channel 15
//     Task_P1 Outputs/IO.Q202[16] <-> Q202 (GSIO-A-16DON)/Digital Outputs/Channel 16
//     Task_P1 Outputs/IO.Q202[1] <-> Q202 (GSIO-A-16DON)/Digital Outputs/Channel 1
//     Task_P1 Outputs/IO.Q202[2] <-> Q202 (GSIO-A-16DON)/Digital Outputs/Channel 2
//     Task_P1 Outputs/IO.Q202[3] <-> Q202 (GSIO-A-16DON)/Digital Outputs/Channel 3
//     Task_P1 Outputs/IO.Q202[4] <-> Q202 (GSIO-A-16DON)/Digital Outputs/Channel 4
//     Task_P1 Outputs/IO.Q202[5] <-> Q202 (GSIO-A-16DON)/Digital Outputs/Channel 5
//     Task_P1 Outputs/IO.Q202[6] <-> Q202 (GSIO-A-16DON)/Digital Outputs/Channel 6
//     Task_P1 Outputs/IO.Q202[7] <-> Q202 (GSIO-A-16DON)/Digital Outputs/Channel 7
//     Task_P1 Outputs/IO.Q202[8] <-> Q202 (GSIO-A-16DON)/Digital Outputs/Channel 8
//     Task_P1 Outputs/IO.Q202[9] <-> Q202 (GSIO-A-16DON)/Digital Outputs/Channel 9
//     Task_P1 Outputs/IO.Q203[10] <-> Q203 (GSIO-A-16DON)/Digital Outputs/Channel 10
//     Task_P1 Outputs/IO.Q203[11] <-> Q203 (GSIO-A-16DON)/Digital Outputs/Channel 11
//     Task_P1 Outputs/IO.Q203[12] <-> Q203 (GSIO-A-16DON)/Digital Outputs/Channel 12
//     Task_P1 Outputs/IO.Q203[13] <-> Q203 (GSIO-A-16DON)/Digital Outputs/Channel 13
//     Task_P1 Outputs/IO.Q203[14] <-> Q203 (GSIO-A-16DON)/Digital Outputs/Channel 14
//     Task_P1 Outputs/IO.Q203[15] <-> Q203 (GSIO-A-16DON)/Digital Outputs/Channel 15
//     Task_P1 Outputs/IO.Q203[16] <-> Q203 (GSIO-A-16DON)/Digital Outputs/Channel 16
//     Task_P1 Outputs/IO.Q203[1] <-> Q203 (GSIO-A-16DON)/Digital Outputs/Channel 1
//     Task_P1 Outputs/IO.Q203[2] <-> Q203 (GSIO-A-16DON)/Digital Outputs/Channel 2
//     Task_P1 Outputs/IO.Q203[3] <-> Q203 (GSIO-A-16DON)/Digital Outputs/Channel 3
//     Task_P1 Outputs/IO.Q203[4] <-> Q203 (GSIO-A-16DON)/Digital Outputs/Channel 4
//     Task_P1 Outputs/IO.Q203[5] <-> Q203 (GSIO-A-16DON)/Digital Outputs/Channel 5
//     Task_P1 Outputs/IO.Q203[6] <-> Q203 (GSIO-A-16DON)/Digital Outputs/Channel 6
//     Task_P1 Outputs/IO.Q203[7] <-> Q203 (GSIO-A-16DON)/Digital Outputs/Channel 7
//     Task_P1 Outputs/IO.Q203[8] <-> Q203 (GSIO-A-16DON)/Digital Outputs/Channel 8
//     Task_P1 Outputs/IO.Q203[9] <-> Q203 (GSIO-A-16DON)/Digital Outputs/Channel 9
//     Task_P1 Outputs/IO.Q204[10] <-> Q204 (GSIO-A-16DON)/Digital Outputs/Channel 10
//     Task_P1 Outputs/IO.Q204[11] <-> Q204 (GSIO-A-16DON)/Digital Outputs/Channel 11
//     Task_P1 Outputs/IO.Q204[12] <-> Q204 (GSIO-A-16DON)/Digital Outputs/Channel 12
//     Task_P1 Outputs/IO.Q204[13] <-> Q204 (GSIO-A-16DON)/Digital Outputs/Channel 13
//     Task_P1 Outputs/IO.Q204[14] <-> Q204 (GSIO-A-16DON)/Digital Outputs/Channel 14
//     Task_P1 Outputs/IO.Q204[15] <-> Q204 (GSIO-A-16DON)/Digital Outputs/Channel 15
//     Task_P1 Outputs/IO.Q204[16] <-> Q204 (GSIO-A-16DON)/Digital Outputs/Channel 16
//     Task_P1 Outputs/IO.Q204[1] <-> Q204 (GSIO-A-16DON)/Digital Outputs/Channel 1
//     Task_P1 Outputs/IO.Q204[2] <-> Q204 (GSIO-A-16DON)/Digital Outputs/Channel 2
//     Task_P1 Outputs/IO.Q204[3] <-> Q204 (GSIO-A-16DON)/Digital Outputs/Channel 3
//     Task_P1 Outputs/IO.Q204[4] <-> Q204 (GSIO-A-16DON)/Digital Outputs/Channel 4
//     Task_P1 Outputs/IO.Q204[5] <-> Q204 (GSIO-A-16DON)/Digital Outputs/Channel 5
//     Task_P1 Outputs/IO.Q204[6] <-> Q204 (GSIO-A-16DON)/Digital Outputs/Channel 6
//     Task_P1 Outputs/IO.Q204[7] <-> Q204 (GSIO-A-16DON)/Digital Outputs/Channel 7
//     Task_P1 Outputs/IO.Q204[8] <-> Q204 (GSIO-A-16DON)/Digital Outputs/Channel 8
//     Task_P1 Outputs/IO.Q204[9] <-> Q204 (GSIO-A-16DON)/Digital Outputs/Channel 9
//     Task_P1 Outputs/IO.Q205[10] <-> Q205 (GSIO-A-16DON)/Digital Outputs/Channel 10
//     Task_P1 Outputs/IO.Q205[11] <-> Q205 (GSIO-A-16DON)/Digital Outputs/Channel 11
//     Task_P1 Outputs/IO.Q205[12] <-> Q205 (GSIO-A-16DON)/Digital Outputs/Channel 12
//     Task_P1 Outputs/IO.Q205[13] <-> Q205 (GSIO-A-16DON)/Digital Outputs/Channel 13
//     Task_P1 Outputs/IO.Q205[14] <-> Q205 (GSIO-A-16DON)/Digital Outputs/Channel 14
//     Task_P1 Outputs/IO.Q205[15] <-> Q205 (GSIO-A-16DON)/Digital Outputs/Channel 15
//     Task_P1 Outputs/IO.Q205[16] <-> Q205 (GSIO-A-16DON)/Digital Outputs/Channel 16
//     Task_P1 Outputs/IO.Q205[1] <-> Q205 (GSIO-A-16DON)/Digital Outputs/Channel 1
//     Task_P1 Outputs/IO.Q205[2] <-> Q205 (GSIO-A-16DON)/Digital Outputs/Channel 2
//     Task_P1 Outputs/IO.Q205[3] <-> Q205 (GSIO-A-16DON)/Digital Outputs/Channel 3
//     Task_P1 Outputs/IO.Q205[4] <-> Q205 (GSIO-A-16DON)/Digital Outputs/Channel 4
//     Task_P1 Outputs/IO.Q205[5] <-> Q205 (GSIO-A-16DON)/Digital Outputs/Channel 5
//     Task_P1 Outputs/IO.Q205[6] <-> Q205 (GSIO-A-16DON)/Digital Outputs/Channel 6
//     Task_P1 Outputs/IO.Q205[7] <-> Q205 (GSIO-A-16DON)/Digital Outputs/Channel 7
//     Task_P1 Outputs/IO.Q205[8] <-> Q205 (GSIO-A-16DON)/Digital Outputs/Channel 8
//     Task_P1 Outputs/IO.Q205[9] <-> Q205 (GSIO-A-16DON)/Digital Outputs/Channel 9
//     Task_P1 Outputs/IO.Q206[10] <-> Q206 (GSIO-A-16DON)/Digital Outputs/Channel 10
//     Task_P1 Outputs/IO.Q206[11] <-> Q206 (GSIO-A-16DON)/Digital Outputs/Channel 11
//     Task_P1 Outputs/IO.Q206[12] <-> Q206 (GSIO-A-16DON)/Digital Outputs/Channel 12
//     Task_P1 Outputs/IO.Q206[13] <-> Q206 (GSIO-A-16DON)/Digital Outputs/Channel 13
//     Task_P1 Outputs/IO.Q206[14] <-> Q206 (GSIO-A-16DON)/Digital Outputs/Channel 14
//     Task_P1 Outputs/IO.Q206[15] <-> Q206 (GSIO-A-16DON)/Digital Outputs/Channel 15
//     Task_P1 Outputs/IO.Q206[16] <-> Q206 (GSIO-A-16DON)/Digital Outputs/Channel 16
//     Task_P1 Outputs/IO.Q206[1] <-> Q206 (GSIO-A-16DON)/Digital Outputs/Channel 1
//     Task_P1 Outputs/IO.Q206[2] <-> Q206 (GSIO-A-16DON)/Digital Outputs/Channel 2
//     Task_P1 Outputs/IO.Q206[3] <-> Q206 (GSIO-A-16DON)/Digital Outputs/Channel 3
//     Task_P1 Outputs/IO.Q206[4] <-> Q206 (GSIO-A-16DON)/Digital Outputs/Channel 4
//     Task_P1 Outputs/IO.Q206[5] <-> Q206 (GSIO-A-16DON)/Digital Outputs/Channel 5
//     Task_P1 Outputs/IO.Q206[6] <-> Q206 (GSIO-A-16DON)/Digital Outputs/Channel 6
//     Task_P1 Outputs/IO.Q206[7] <-> Q206 (GSIO-A-16DON)/Digital Outputs/Channel 7
//     Task_P1 Outputs/IO.Q206[8] <-> Q206 (GSIO-A-16DON)/Digital Outputs/Channel 8
//     Task_P1 Outputs/IO.Q206[9] <-> Q206 (GSIO-A-16DON)/Digital Outputs/Channel 9
//     Task_P1 Outputs/IO.Q207[10] <-> Q207 (GSIO-A-16DON)/Digital Outputs/Channel 10
//     Task_P1 Outputs/IO.Q207[11] <-> Q207 (GSIO-A-16DON)/Digital Outputs/Channel 11
//     Task_P1 Outputs/IO.Q207[12] <-> Q207 (GSIO-A-16DON)/Digital Outputs/Channel 12
//     Task_P1 Outputs/IO.Q207[13] <-> Q207 (GSIO-A-16DON)/Digital Outputs/Channel 13
//     Task_P1 Outputs/IO.Q207[14] <-> Q207 (GSIO-A-16DON)/Digital Outputs/Channel 14
//     Task_P1 Outputs/IO.Q207[15] <-> Q207 (GSIO-A-16DON)/Digital Outputs/Channel 15
//     Task_P1 Outputs/IO.Q207[16] <-> Q207 (GSIO-A-16DON)/Digital Outputs/Channel 16
//     Task_P1 Outputs/IO.Q207[1] <-> Q207 (GSIO-A-16DON)/Digital Outputs/Channel 1
//     Task_P1 Outputs/IO.Q207[2] <-> Q207 (GSIO-A-16DON)/Digital Outputs/Channel 2
//     Task_P1 Outputs/IO.Q207[3] <-> Q207 (GSIO-A-16DON)/Digital Outputs/Channel 3
//     Task_P1 Outputs/IO.Q207[4] <-> Q207 (GSIO-A-16DON)/Digital Outputs/Channel 4
//     Task_P1 Outputs/IO.Q207[5] <-> Q207 (GSIO-A-16DON)/Digital Outputs/Channel 5
//     Task_P1 Outputs/IO.Q207[6] <-> Q207 (GSIO-A-16DON)/Digital Outputs/Channel 6
//     Task_P1 Outputs/IO.Q207[7] <-> Q207 (GSIO-A-16DON)/Digital Outputs/Channel 7
//     Task_P1 Outputs/IO.Q207[8] <-> Q207 (GSIO-A-16DON)/Digital Outputs/Channel 8
//     Task_P1 Outputs/IO.Q207[9] <-> Q207 (GSIO-A-16DON)/Digital Outputs/Channel 9
//     Task_P1 Outputs/IO.Q208[10] <-> Q208 (GSIO-A-16DON)/Digital Outputs/Channel 10
//     Task_P1 Outputs/IO.Q208[11] <-> Q208 (GSIO-A-16DON)/Digital Outputs/Channel 11
//     Task_P1 Outputs/IO.Q208[12] <-> Q208 (GSIO-A-16DON)/Digital Outputs/Channel 12
//     Task_P1 Outputs/IO.Q208[13] <-> Q208 (GSIO-A-16DON)/Digital Outputs/Channel 13
//     Task_P1 Outputs/IO.Q208[14] <-> Q208 (GSIO-A-16DON)/Digital Outputs/Channel 14
//     Task_P1 Outputs/IO.Q208[15] <-> Q208 (GSIO-A-16DON)/Digital Outputs/Channel 15
//     Task_P1 Outputs/IO.Q208[16] <-> Q208 (GSIO-A-16DON)/Digital Outputs/Channel 16
//     Task_P1 Outputs/IO.Q208[1] <-> Q208 (GSIO-A-16DON)/Digital Outputs/Channel 1
//     Task_P1 Outputs/IO.Q208[2] <-> Q208 (GSIO-A-16DON)/Digital Outputs/Channel 2
//     Task_P1 Outputs/IO.Q208[3] <-> Q208 (GSIO-A-16DON)/Digital Outputs/Channel 3
//     Task_P1 Outputs/IO.Q208[4] <-> Q208 (GSIO-A-16DON)/Digital Outputs/Channel 4
//     Task_P1 Outputs/IO.Q208[5] <-> Q208 (GSIO-A-16DON)/Digital Outputs/Channel 5
//     Task_P1 Outputs/IO.Q208[6] <-> Q208 (GSIO-A-16DON)/Digital Outputs/Channel 6
//     Task_P1 Outputs/IO.Q208[7] <-> Q208 (GSIO-A-16DON)/Digital Outputs/Channel 7
//     Task_P1 Outputs/IO.Q208[8] <-> Q208 (GSIO-A-16DON)/Digital Outputs/Channel 8
//     Task_P1 Outputs/IO.Q208[9] <-> Q208 (GSIO-A-16DON)/Digital Outputs/Channel 9
//     Task_P1 Outputs/IO.Q209[10] <-> Q209 (GSIO-A-16DON)/Digital Outputs/Channel 10
//     Task_P1 Outputs/IO.Q209[11] <-> Q209 (GSIO-A-16DON)/Digital Outputs/Channel 11
//     Task_P1 Outputs/IO.Q209[12] <-> Q209 (GSIO-A-16DON)/Digital Outputs/Channel 12
//     Task_P1 Outputs/IO.Q209[13] <-> Q209 (GSIO-A-16DON)/Digital Outputs/Channel 13
//     Task_P1 Outputs/IO.Q209[14] <-> Q209 (GSIO-A-16DON)/Digital Outputs/Channel 14
//     Task_P1 Outputs/IO.Q209[15] <-> Q209 (GSIO-A-16DON)/Digital Outputs/Channel 15
//     Task_P1 Outputs/IO.Q209[16] <-> Q209 (GSIO-A-16DON)/Digital Outputs/Channel 16
//     Task_P1 Outputs/IO.Q209[1] <-> Q209 (GSIO-A-16DON)/Digital Outputs/Channel 1
//     Task_P1 Outputs/IO.Q209[2] <-> Q209 (GSIO-A-16DON)/Digital Outputs/Channel 2
//     Task_P1 Outputs/IO.Q209[3] <-> Q209 (GSIO-A-16DON)/Digital Outputs/Channel 3
//     Task_P1 Outputs/IO.Q209[4] <-> Q209 (GSIO-A-16DON)/Digital Outputs/Channel 4
//     Task_P1 Outputs/IO.Q209[5] <-> Q209 (GSIO-A-16DON)/Digital Outputs/Channel 5
//     Task_P1 Outputs/IO.Q209[6] <-> Q209 (GSIO-A-16DON)/Digital Outputs/Channel 6
//     Task_P1 Outputs/IO.Q209[7] <-> Q209 (GSIO-A-16DON)/Digital Outputs/Channel 7
//     Task_P1 Outputs/IO.Q209[8] <-> Q209 (GSIO-A-16DON)/Digital Outputs/Channel 8
//     Task_P1 Outputs/IO.Q209[9] <-> Q209 (GSIO-A-16DON)/Digital Outputs/Channel 9
//   MQPLC/MQPLC Instance <-> Device 3 (EtherCAT)/P2M1正极送料分段皮带1[20(模切)] (InoSV660N)
//     Task_P1 Inputs/GMotion.arrAxisCtrl[20].Io.ErrorCode <-> Inputs/Error code
//     Task_P1 Inputs/GMotion.iActTorque_M[20] <-> Inputs/Torque actual value
//   MQPLC/MQPLC Instance <-> Device 3 (EtherCAT)/P2M1负极送料分段皮带1[44（模切）] (InoSV660N)
//     Task_P1 Inputs/GMotion.arrAxisCtrl[44].Io.ErrorCode <-> Inputs/Error code
//     Task_P1 Inputs/GMotion.iActTorque_M[44] <-> Inputs/Torque actual value
//   MQPLC/MQPLC Instance <-> NC-Task 1 SAF/Axes/Axis001_1 P1An_UnWind_L
//     Task_P1 Inputs/GMotion.arrAxis[1].NcToPlc <-> Outputs/ToPlc
//     Task_P1 Outputs/GMotion.arrAxis[1].PlcToNc <-> Inputs/FromPlc
//   MQPLC/MQPLC Instance <-> NC-Task 1 SAF/Axes/Axis002_2 P1An_UnWind_R
//     Task_P1 Inputs/GMotion.arrAxis[2].NcToPlc <-> Outputs/ToPlc
//     Task_P1 Outputs/GMotion.arrAxis[2].PlcToNc <-> Inputs/FromPlc
//   MQPLC/MQPLC Instance <-> NC-Task 1 SAF/Axes/Axis003_3 P1An_PoleTension
//     Task_P1 Inputs/GMotion.arrAxis[3].NcToPlc <-> Outputs/ToPlc
//     Task_P1 Outputs/GMotion.arrAxis[3].PlcToNc <-> Inputs/FromPlc
//   MQPLC/MQPLC Instance <-> NC-Task 1 SAF/Axes/Axis004_4 P1An_DriverAux
//     Task_P1 Inputs/GMotion.arrAxis[4].NcToPlc <-> Outputs/ToPlc
//     Task_P1 Outputs/GMotion.arrAxis[4].PlcToNc <-> Inputs/FromPlc
//   MQPLC/MQPLC Instance <-> NC-Task 1 SAF/Axes/Axis005_5 P1An_BuffeLine
//     Task_P1 Inputs/GMotion.arrAxis[5].NcToPlc <-> Outputs/ToPlc
//     Task_P1 Outputs/GMotion.arrAxis[5].PlcToNc <-> Inputs/FromPlc
//   MQPLC/MQPLC Instance <-> NC-Task 1 SAF/Axes/Axis006_6 P1An_Mould
//     Task_P1 Inputs/GMotion.arrAxis[6].NcToPlc <-> Outputs/ToPlc
//     Task_P1 Outputs/GMotion.arrAxis[6].PlcToNc <-> Inputs/FromPlc
//   MQPLC/MQPLC Instance <-> NC-Task 1 SAF/Axes/Axis007_7 P1An_MouldRectify_X
//     Task_P1 Inputs/GMotion.arrAxis[7].NcToPlc <-> Outputs/ToPlc
//     Task_P1 Outputs/GMotion.arrAxis[7].PlcToNc <-> Inputs/FromPlc
//   MQPLC/MQPLC Instance <-> NC-Task 1 SAF/Axes/Axis008_8 P1An_MouldRectify_Y
//     Task_P1 Inputs/GMotion.arrAxis[8].NcToPlc <-> Outputs/ToPlc
//     Task_P1 Outputs/GMotion.arrAxis[8].PlcToNc <-> Inputs/FromPlc
//   MQPLC/MQPLC Instance <-> NC-Task 1 SAF/Axes/Axis009_9 P1An_DriverDDR
//     Task_P1 Inputs/GMotion.arrAxis[9].NcToPlc <-> Outputs/ToPlc
//     Task_P1 Outputs/GMotion.arrAxis[9].PlcToNc <-> Inputs/FromPlc
//   MQPLC/MQPLC Instance <-> NC-Task 1 SAF/Axes/Axis010_10 P1An_Cuter
//     Task_P1 Inputs/GMotion.arrAxis[10].NcToPlc <-> Outputs/ToPlc
//     Task_P1 Outputs/GMotion.arrAxis[10].PlcToNc <-> Inputs/FromPlc
//   MQPLC/MQPLC Instance <-> NC-Task 1 SAF/Axes/Axis011_11 P1An_CuterDegRectify
//     Task_P1 Inputs/GMotion.arrAxis[11].NcToPlc <-> Outputs/ToPlc
//     Task_P1 Outputs/GMotion.arrAxis[11].PlcToNc <-> Inputs/FromPlc
//   MQPLC/MQPLC Instance <-> NC-Task 1 SAF/Axes/Axis012_12 P1An_CuterBelt
//     Task_P1 Inputs/GMotion.arrAxis[12].NcToPlc <-> Outputs/ToPlc
//     Task_P1 Outputs/GMotion.arrAxis[12].PlcToNc <-> Inputs/FromPlc
//   MQPLC/MQPLC Instance <-> NC-Task 1 SAF/Axes/Axis013_13 P1An_CuterBeltChange
//     Task_P1 Inputs/GMotion.arrAxis[13].NcToPlc <-> Outputs/ToPlc
//     Task_P1 Outputs/GMotion.arrAxis[13].PlcToNc <-> Inputs/FromPlc
//   MQPLC/MQPLC Instance <-> NC-Task 1 SAF/Axes/Axis014_14 P1An_CCDPressPush
//     Task_P1 Inputs/GMotion.arrAxis[14].NcToPlc <-> Outputs/ToPlc
//     Task_P1 Outputs/GMotion.arrAxis[14].PlcToNc <-> Inputs/FromPlc
//   MQPLC/MQPLC Instance <-> NC-Task 1 SAF/Axes/Axis015_15 P1An_NGPushReverseBelt
//     Task_P1 Inputs/GMotion.arrAxis[15].NcToPlc <-> Outputs/ToPlc
//     Task_P1 Outputs/GMotion.arrAxis[15].PlcToNc <-> Inputs/FromPlc
//   MQPLC/MQPLC Instance <-> NC-Task 1 SAF/Axes/Axis016_16 P1An_NGPush1
//     Task_P1 Inputs/GMotion.arrAxis[16].NcToPlc <-> Outputs/ToPlc
//     Task_P1 Outputs/GMotion.arrAxis[16].PlcToNc <-> Inputs/FromPlc
//   MQPLC/MQPLC Instance <-> NC-Task 1 SAF/Axes/Axis017_17 P1An_NGPush2
//     Task_P1 Inputs/GMotion.arrAxis[17].NcToPlc <-> Outputs/ToPlc
//     Task_P1 Outputs/GMotion.arrAxis[17].PlcToNc <-> Inputs/FromPlc
//   MQPLC/MQPLC Instance <-> NC-Task 1 SAF/Axes/Axis018_18 P1An_DedustBelt
//     Task_P1 Inputs/GMotion.arrAxis[18].NcToPlc <-> Outputs/ToPlc
//     Task_P1 Outputs/GMotion.arrAxis[18].PlcToNc <-> Inputs/FromPlc
//   MQPLC/MQPLC Instance <-> NC-Task 1 SAF/Axes/Axis019_19 P1An_DedustReverseBelt
//     Task_P1 Inputs/GMotion.arrAxis[19].NcToPlc <-> Outputs/ToPlc
//     Task_P1 Outputs/GMotion.arrAxis[19].PlcToNc <-> Inputs/FromPlc
//   MQPLC/MQPLC Instance <-> NC-Task 1 SAF/Axes/Axis020_20 P1An_SubBelt1
//     Task_P1 Inputs/GMotion.arrAxis[20].NcToPlc <-> Outputs/ToPlc
//     Task_P1 Outputs/GMotion.arrAxis[20].PlcToNc <-> Inputs/FromPlc
//   MQPLC/MQPLC Instance <-> NC-Task 1 SAF/Axes/Axis021_21 P1An_SubBelt2
//     Task_P1 Inputs/GMotion.arrAxis[21].NcToPlc <-> Outputs/ToPlc
//     Task_P1 Outputs/GMotion.arrAxis[21].PlcToNc <-> Inputs/FromPlc
//   MQPLC/MQPLC Instance <-> NC-Task 1 SAF/Axes/Axis022_22 P1An_SubBelt3
//     Task_P1 Inputs/GMotion.arrAxis[22].NcToPlc <-> Outputs/ToPlc
//     Task_P1 Outputs/GMotion.arrAxis[22].PlcToNc <-> Inputs/FromPlc
//   MQPLC/MQPLC Instance <-> NC-Task 1 SAF/Axes/Axis023_23 P1An_Ready1
//     Task_P1 Inputs/GMotion.arrAxis[23].NcToPlc <-> Outputs/ToPlc
//     Task_P1 Outputs/GMotion.arrAxis[23].PlcToNc <-> Inputs/FromPlc
//   MQPLC/MQPLC Instance <-> NC-Task 1 SAF/Axes/Axis024_24 P1An_Ready2
//     Task_P1 Inputs/GMotion.arrAxis[24].NcToPlc <-> Outputs/ToPlc
//     Task_P1 Outputs/GMotion.arrAxis[24].PlcToNc <-> Inputs/FromPlc
//   MQPLC/MQPLC Instance <-> NC-Task 1 SAF/Axes/Axis025_25 P1Ca_UnWind_L
//     Task_P1 Inputs/GMotion.arrAxis[25].NcToPlc <-> Outputs/ToPlc
//     Task_P1 Outputs/GMotion.arrAxis[25].PlcToNc <-> Inputs/FromPlc
//   MQPLC/MQPLC Instance <-> NC-Task 1 SAF/Axes/Axis026_26 P1Ca_UnWind_R
//     Task_P1 Inputs/GMotion.arrAxis[26].NcToPlc <-> Outputs/ToPlc
//     Task_P1 Outputs/GMotion.arrAxis[26].PlcToNc <-> Inputs/FromPlc
//   MQPLC/MQPLC Instance <-> NC-Task 1 SAF/Axes/Axis027_27 P1Ca_PoleTension
//     Task_P1 Inputs/GMotion.arrAxis[27].NcToPlc <-> Outputs/ToPlc
//     Task_P1 Outputs/GMotion.arrAxis[27].PlcToNc <-> Inputs/FromPlc
//   MQPLC/MQPLC Instance <-> NC-Task 1 SAF/Axes/Axis028_28 P1Ca_DriverAux
//     Task_P1 Inputs/GMotion.arrAxis[28].NcToPlc <-> Outputs/ToPlc
//     Task_P1 Outputs/GMotion.arrAxis[28].PlcToNc <-> Inputs/FromPlc
//   MQPLC/MQPLC Instance <-> NC-Task 1 SAF/Axes/Axis029_29 P1Ca_BuffeLine
//     Task_P1 Inputs/GMotion.arrAxis[29].NcToPlc <-> Outputs/ToPlc
//     Task_P1 Outputs/GMotion.arrAxis[29].PlcToNc <-> Inputs/FromPlc
//   MQPLC/MQPLC Instance <-> NC-Task 1 SAF/Axes/Axis030_30 P1Ca_Mould
//     Task_P1 Inputs/GMotion.arrAxis[30].NcToPlc <-> Outputs/ToPlc
//     Task_P1 Outputs/GMotion.arrAxis[30].PlcToNc <-> Inputs/FromPlc
//   MQPLC/MQPLC Instance <-> NC-Task 1 SAF/Axes/Axis031_31 P1Ca_MouldRectify_X
//     Task_P1 Inputs/GMotion.arrAxis[31].NcToPlc <-> Outputs/ToPlc
//     Task_P1 Outputs/GMotion.arrAxis[31].PlcToNc <-> Inputs/FromPlc
//   MQPLC/MQPLC Instance <-> NC-Task 1 SAF/Axes/Axis032_32 P1Ca_MouldRectify_Y
//     Task_P1 Inputs/GMotion.arrAxis[32].NcToPlc <-> Outputs/ToPlc
//     Task_P1 Outputs/GMotion.arrAxis[32].PlcToNc <-> Inputs/FromPlc
//   MQPLC/MQPLC Instance <-> NC-Task 1 SAF/Axes/Axis033_33 P1Ca_DriverDDR
//     Task_P1 Inputs/GMotion.arrAxis[33].NcToPlc <-> Outputs/ToPlc
//     Task_P1 Outputs/GMotion.arrAxis[33].PlcToNc <-> Inputs/FromPlc
//   MQPLC/MQPLC Instance <-> NC-Task 1 SAF/Axes/Axis034_34 P1Ca_Cuter
//     Task_P1 Inputs/GMotion.arrAxis[34].NcToPlc <-> Outputs/ToPlc
//     Task_P1 Outputs/GMotion.arrAxis[34].PlcToNc <-> Inputs/FromPlc
//   MQPLC/MQPLC Instance <-> NC-Task 1 SAF/Axes/Axis035_35 P1Ca_CuterDegRectify
//     Task_P1 Inputs/GMotion.arrAxis[35].NcToPlc <-> Outputs/ToPlc
//     Task_P1 Outputs/GMotion.arrAxis[35].PlcToNc <-> Inputs/FromPlc
//   MQPLC/MQPLC Instance <-> NC-Task 1 SAF/Axes/Axis036_36 P1Ca_CuterBelt
//     Task_P1 Inputs/GMotion.arrAxis[36].NcToPlc <-> Outputs/ToPlc
//     Task_P1 Outputs/GMotion.arrAxis[36].PlcToNc <-> Inputs/FromPlc
//   MQPLC/MQPLC Instance <-> NC-Task 1 SAF/Axes/Axis037_37 P1Ca_CuterBeltChange
//     Task_P1 Inputs/GMotion.arrAxis[37].NcToPlc <-> Outputs/ToPlc
//     Task_P1 Outputs/GMotion.arrAxis[37].PlcToNc <-> Inputs/FromPlc
//   MQPLC/MQPLC Instance <-> NC-Task 1 SAF/Axes/Axis038_38 P1Ca_CCDPressPush
//     Task_P1 Inputs/GMotion.arrAxis[38].NcToPlc <-> Outputs/ToPlc
//     Task_P1 Outputs/GMotion.arrAxis[38].PlcToNc <-> Inputs/FromPlc
//   MQPLC/MQPLC Instance <-> NC-Task 1 SAF/Axes/Axis039_39 P1Ca_NGPushReverseBelt
//     Task_P1 Inputs/GMotion.arrAxis[39].NcToPlc <-> Outputs/ToPlc
//     Task_P1 Outputs/GMotion.arrAxis[39].PlcToNc <-> Inputs/FromPlc
//   MQPLC/MQPLC Instance <-> NC-Task 1 SAF/Axes/Axis040_40 P1Ca_NGPush1
//     Task_P1 Inputs/GMotion.arrAxis[40].NcToPlc <-> Outputs/ToPlc
//     Task_P1 Outputs/GMotion.arrAxis[40].PlcToNc <-> Inputs/FromPlc
//   MQPLC/MQPLC Instance <-> NC-Task 1 SAF/Axes/Axis041_41 P1Ca_NGPush2
//     Task_P1 Inputs/GMotion.arrAxis[41].NcToPlc <-> Outputs/ToPlc
//     Task_P1 Outputs/GMotion.arrAxis[41].PlcToNc <-> Inputs/FromPlc
//   MQPLC/MQPLC Instance <-> NC-Task 1 SAF/Axes/Axis042_42 P1Ca_DedustBelt
//     Task_P1 Inputs/GMotion.arrAxis[42].NcToPlc <-> Outputs/ToPlc
//     Task_P1 Outputs/GMotion.arrAxis[42].PlcToNc <-> Inputs/FromPlc
//   MQPLC/MQPLC Instance <-> NC-Task 1 SAF/Axes/Axis043_43 P1Ca_DedustReverseBelt
//     Task_P1 Inputs/GMotion.arrAxis[43].NcToPlc <-> Outputs/ToPlc
//     Task_P1 Outputs/GMotion.arrAxis[43].PlcToNc <-> Inputs/FromPlc
//   MQPLC/MQPLC Instance <-> NC-Task 1 SAF/Axes/Axis044_44 P1Ca_SubBelt1
//     Task_P1 Inputs/GMotion.arrAxis[44].NcToPlc <-> Outputs/ToPlc
//     Task_P1 Outputs/GMotion.arrAxis[44].PlcToNc <-> Inputs/FromPlc
//   MQPLC/MQPLC Instance <-> NC-Task 1 SAF/Axes/Axis045_45 P1Ca_SubBelt2
//     Task_P1 Inputs/GMotion.arrAxis[45].NcToPlc <-> Outputs/ToPlc
//     Task_P1 Outputs/GMotion.arrAxis[45].PlcToNc <-> Inputs/FromPlc
//   MQPLC/MQPLC Instance <-> NC-Task 1 SAF/Axes/Axis046_46 P1Ca_SubBelt3
//     Task_P1 Inputs/GMotion.arrAxis[46].NcToPlc <-> Outputs/ToPlc
//     Task_P1 Outputs/GMotion.arrAxis[46].PlcToNc <-> Inputs/FromPlc
//   MQPLC/MQPLC Instance <-> NC-Task 1 SAF/Axes/Axis047_47 P1Ca_Ready1
//     Task_P1 Inputs/GMotion.arrAxis[47].NcToPlc <-> Outputs/ToPlc
//     Task_P1 Outputs/GMotion.arrAxis[47].PlcToNc <-> Inputs/FromPlc
//   MQPLC/MQPLC Instance <-> NC-Task 1 SAF/Axes/Axis048_48 P1Ca_Ready2
//     Task_P1 Inputs/GMotion.arrAxis[48].NcToPlc <-> Outputs/ToPlc
//     Task_P1 Outputs/GMotion.arrAxis[48].PlcToNc <-> Inputs/FromPlc
//   MQPLC/MQPLC Instance <-> NC-Task 1 SAF/Axes/Axis210_50 P1_VirTimeWind
//     Task_P1 Inputs/GMotion.arrAxis[50].NcToPlc <-> Outputs/ToPlc
//     Task_P1 Outputs/GMotion.arrAxis[50].PlcToNc <-> Inputs/FromPlc
//   MQPLC/MQPLC Instance <-> NC-Task 1 SAF/Axes/Axis211_51 P1An_VirMain
//     Task_P1 Inputs/GMotion.arrAxis[51].NcToPlc <-> Outputs/ToPlc
//     Task_P1 Outputs/GMotion.arrAxis[51].PlcToNc <-> Inputs/FromPlc
//   MQPLC/MQPLC Instance <-> NC-Task 1 SAF/Axes/Axis212_52 P1An_VirDriver
//     Task_P1 Inputs/GMotion.arrAxis[52].NcToPlc <-> Outputs/ToPlc
//     Task_P1 Outputs/GMotion.arrAxis[52].PlcToNc <-> Inputs/FromPlc
//   MQPLC/MQPLC Instance <-> NC-Task 1 SAF/Axes/Axis213_53 P1An_VirBelt
//     Task_P1 Inputs/GMotion.arrAxis[53].NcToPlc <-> Outputs/ToPlc
//     Task_P1 Outputs/GMotion.arrAxis[53].PlcToNc <-> Inputs/FromPlc
//   MQPLC/MQPLC Instance <-> NC-Task 1 SAF/Axes/Axis214_56 P1Ca_VirMain
//     Task_P1 Inputs/GMotion.arrAxis[56].NcToPlc <-> Outputs/ToPlc
//     Task_P1 Outputs/GMotion.arrAxis[56].PlcToNc <-> Inputs/FromPlc
//   MQPLC/MQPLC Instance <-> NC-Task 1 SAF/Axes/Axis215_57 P1Ca_VirDriver
//     Task_P1 Inputs/GMotion.arrAxis[57].NcToPlc <-> Outputs/ToPlc
//     Task_P1 Outputs/GMotion.arrAxis[57].PlcToNc <-> Inputs/FromPlc
//   MQPLC/MQPLC Instance <-> NC-Task 1 SAF/Axes/Axis216_58 P1Ca_VirBelt
//     Task_P1 Inputs/GMotion.arrAxis[58].NcToPlc <-> Outputs/ToPlc
//     Task_P1 Outputs/GMotion.arrAxis[58].PlcToNc <-> Inputs/FromPlc

CONFIGURATION MQPLC
    RESOURCE PLC ON TwinCAT3
        TASK Task_P1(INTERVAL := T#2ms, PRIORITY := 8);
        PROGRAM MAIN WITH Task_P1 : MAIN;
    END_RESOURCE
END_CONFIGURATION

// ---- DUTs/01_AxisCO_Ntrol/ST_ECYCtrl.TcDUT
TYPE ST_ECYCtrl :
STRUCT
    bServON   :BOOL;   
    bHome      :BOOL;   
    bReset      :BOOL;   
    bStop         :BOOL;   
   bJog_P         :BOOL;   
   bJog_N        :BOOL;   
   Pos_Start      :BOOL;   
   fTagetPos     :REAL;
   fVel:           REAL;
   fAcc        :REAL;  
   fDec        :REAL;  
  // Delay_Time  :TIME;


     bHomed         :BOOL; 
     Pos_Done       :BOOL;   //定位完成
     Home_Alm      :BOOL;  //回零超时报警
     Pos_Alm         :BOOL; //定位超时报警



END_STRUCT
END_TYPE

// ---- DUTs/01_AxisCO_Ntrol/ST_JXCE.TcDUT
TYPE ST_JXCE :
STRUCT
      out_Control             AT  %Q*  :     UINT;  // 电机控制
      out_Function            AT  %Q*  :    UINT;  // 电机功能
      out_Start                 AT  %Q*  :   USINT;  // 电机启动定位
      out_Mode               AT  %Q*  :   USINT;  // 电机定位模式
      out_Cmd_Vel           AT  %Q*  :    UINT;  // 电机命令速度
      out_Cmd_Pos           AT  %Q*  :   DINT;  // 电机命令位置
      out_Cmd_Acc           AT  %Q*  :   UINT;  // 电机命令加速度
      out_Cmd_Dec          AT  %Q*  :    UINT;  // 电机命令减速度

      in_Status               AT  %I*  :     UINT;  // 电机状态
      in_Flag                 AT  %I*  :     UINT;  // 电机标志位
      in_Act_Pos              AT  %I*  :     DINT;  // 电机反馈位置
      in_Act_Vel             AT  %I*  :     UINT;  // 电机反馈速度
   
     in_Latest_Alm          AT  %I*  :     USINT;  // 电机最新报警

END_STRUCT
END_TYPE

// ---- DUTs/01_AxisCO_Ntrol/ST_DustMotor.TcDUT
TYPE ST_DustMotor :
STRUCT
	bJog_FW			:BOOL;		//手动正转
	bJog_BW			:BOOL;	 //手动反转
	
	bRun_FW			:BOOL;		//正转
	bRun_BW			:BOOL;	 //反转
	
	bo_Pul			:BOOL;		//电机启动
	bo_Dir			:BOOL;//电机方向(0=正转)

END_STRUCT
END_TYPE

// ---- DUTs/01_AxisCO_Ntrol_1/ST_AxisCmd.TcDUT
TYPE ST_AxisCmd :  //轴运动控制相关
STRUCT

   bDynamitcsParSel      :INT:=1;  // 1:NC          2:UserDefine


	bEnable			        :BOOL;				    (*使能*)
	fOverride			    :REAL:=100;			(*MC_power中实际倍率的设定，默认值为100*)
	bEnableFw		        :BOOL:=TRUE;		 (*正向使能*)
	bEnableBw		    :BOOL:=TRUE;	 	(*负向使能*)

	bJog_Fw			    :BOOL;			     	(*正向点动*)
	bJog_Bw			    :BOOL;			    	(*反向点动*)

	bMoveAbs	 	        :BOOL;				    (*运行绝对位置*)
	fPositon_of_Abs	 	:REAL;					(*绝对位置位移*)

	bMoveRel		        :BOOL;				   (*运行当对位置*)
	fPosition_of_Rel	    :REAL;				   (*相对位置位移*)
	
	arrbModuloGo		 :ARRAY[0..10] OF BOOL;	(*运行模长位置*)
	arrbModuloPoint	 :ARRAY[0..10] OF BOOL;	(*模长位置指示*)

	bMoveModulo		 :BOOL;				     (*运行模长位置*)
	fPositon_of_Mod	  :REAL;					  (*模长位置位移*)

	bMoveVelo		    :BOOL;				       (*向一个方向持续运行，方向由前面的正向点动或者反向点动设置*)
	bMoveVeloDir	:MC_Direction := MC_Positive_Direction ;	(*速度运动的方向,MC_Negative_Direction*)

	bHome			       :BOOL;						(*启动回参*)

	bSetPos			       :BOOL;						 (*设置轴当前的位置为一个绝对位置*)
    fSetPos				   :REAL:=0;					(*setpos功能块将轴当前的位置设置为这个变量*)

	iGoSetPos              :INT;                     //GO离散点位_INT
    arrbGoSetPos      :ARRAY[0..10]        OF BOOL;  //GO离散点位_布尔数组
	iRealPoint              :INT;                     //离散点位指示_INIT
    arrbRealPoint        :ARRAY[0..10]        OF BOOL;  //离散点位指示_布尔数组

	bHalt			            :BOOL;				(*暂停*)
	bStop			        :BOOL;				(*停止*)
	bGearOut			    :BOOL;				(*解耦*)
	bReset			        :BOOL;				(*复位*)

	hmiJog_Fw			    :BOOL;				//正向点动_BOOL
	hmibJog_Bw		     :BOOL;				//反向点动_BOOL	
	hmiGoSetPos          :INT;              //GO离散点位_INT


//条件
     Home_Condition       :BOOL;//回原点条件
     JogP_Condition       :BOOL;//点动正转条件
     JogN_Condition       :BOOL;//点动反转条件
     GoPoint_Condition    :ARRAY[0..10] OF BOOL:=[11(TRUE)];//HMI点动定位条件








END_STRUCT
END_TYPE

// ---- DUTs/01_AxisCO_Ntrol_1/ST_AxisCtrl.TcDUT
TYPE ST_AxisCtrl :
STRUCT
    Io                        :ST_AxisIo;  (*轴IO信号*)
    Status                  :ST_AxisStatus;  
    Cmd                    :ST_AxisCmd;  
END_STRUCT
END_TYPE

// ---- DUTs/01_AxisCO_Ntrol_1/ST_AxisIo.TcDUT
TYPE ST_AxisIo :   //轴IO信号
STRUCT

	biNegLimit	             :BOOL;		            (*负限位触发信号*)
	biPosLimit	             :BOOL;		            (*正限位触发信号*)
	biHomeSwitch	     :BOOL;		         (*原点触发信号*)
    DigitalInputs          AT %I*	:  UDINT;
	ErrorCode          AT %I*	:  UINT;//错误代码
END_STRUCT
END_TYPE

// ---- DUTs/01_AxisCO_Ntrol_1/ST_AxisStatus.TcDUT
TYPE ST_AxisStatus :   //轴相关状态
STRUCT

(*status*)
	AxisName		     :STRING(31);		     (*轴名称*)
	AxisID			     :UDINT;		      (*轴在NC中的编号*)
	
    Enabled		         :BOOL;              //使能状态
	Moving              :BOOL;                //轴运行中
	NoMoving          :BOOL;   //轴停止中
    Coupled             :BOOL;   //轴耦合中

	fActPos			     :LREAL;  //轴的当前位置               
	fSetPos			     :LREAL;   //轴的指令位置              
    fModuloActPos		 :REAL;   //轴的当前模长位置             
    fModuloSetPos		 :REAL;      //轴的指令模长位置 
    fActVelo			   :REAL;    //轴的当前速度             
    fSetVelo			   :REAL;    //轴的指令速度
	Homed                :BOOL;        //轴回原点完成          
	Error                   :BOOL;//轴报错
	ErrorID                  :UDINT;//轴报错ID号
    WarningDynamitcsPar    :BOOL; //运动参数警告
	
	bDrivesOP              :BOOL;//驱动器OP状态OK

	
	  ErrorLimitSwitch           :BOOL; //限位报警
END_STRUCT
END_TYPE

// ---- DUTs/01_AxisCO_Ntrol_1/ST_Axis_Par.TcDUT
TYPE ST_Axis_Par ://轴参数
STRUCT
      bLimitSwitchEn          :BOOL;//限位保护开启
	fVelocity_of_Abs	 :REAL:=5;				
	fVelocity_of_Mod	 :REAL:=5;				
	fVelocity_of_Rel	 :REAL:=5;				
	fVelocity_of_Velo	 :REAL:=5;				
	fVelocity_of_Jog	 :REAL:=10;			
	fInchingDistance	 :REAL:=5;				

	arrTargetPoint: ARRAY [0..10] OF REAL;
	//fMaxVelocity:        REAL:=0;	
    fTagatTime                                 :REAL:=0.5;//S  运动时间
    fConVelPercentage                      :REAL:=0.8;//  匀速段占比
    fMaxAccDec                              :LREAL:=50000;//最大加速度
    fMaxVel                                   :LREAL:=2000;//最大速度

	fHomePosition                     :REAL:=10 ;	                          
	fHomeFastSpeed                  :REAL:=20 ;	 
	fHomeSlowSpeed                 :REAL:=10;	 
    HomeLimitDis                       :REAL:=5;	 

	

END_STRUCT
END_TYPE

// ---- DUTs/02_Cylinder/ST_CyCmd.TcDUT
TYPE ST_CyCmd ://
STRUCT
	bON:				        BOOL;	//开关ON
	bOFF:				    BOOL;	//开关OFF
	bFree:				    BOOL;	//泄压

    iType	:	                INT:=1	;	      //气缸类型选择：    1：气缸双控    2：气缸单控        3 电磁阀双控   4 电磁阀单控 
  
	OnCondition:		   BOOL:=TRUE;	//开条件
	OffCondition:		    BOOL:=TRUE;	//关条件
    ErrorTime:		        INT:=5;	

	HMION:	           BOOL;//HMI ON
	HMIOFF:	           BOOL;//HMI OFF


END_STRUCT
END_TYPE

// ---- DUTs/02_Cylinder/ST_CyCtrl.TcDUT
TYPE ST_CyCtrl ://气缸控制UDT  对应单控  双控气缸
STRUCT
   Io           : ST_CYIO;    //气缸IO
   Cmd      :  ST_CyCmd;
   Status     :ST_CyStatus;

END_STRUCT
END_TYPE

// ---- DUTs/02_Cylinder/ST_CYIo.TcDUT
TYPE ST_CYIo ://气缸 I O
STRUCT
	DIOnSwitch:		    BOOL;	//开限位
	DIOFFSwitch:		BOOL;	//关限位

	DOStatus1:          BOOL;//输出状态
	DOStatus2:          BOOL;//输出状态

END_STRUCT
END_TYPE

// ---- DUTs/02_Cylinder/ST_CyStatus.TcDUT
TYPE ST_CyStatus ://
STRUCT
	ONState:	        BOOL;//开状态
	OFFState:	        BOOL;//关状态
	Error1:	            BOOL;//气缸ON报警
	Error2:	            BOOL;//气缸OFF报警
END_STRUCT
END_TYPE

// ---- DUTs/04_Rectify/ST_RecCtrl.TcDUT
TYPE ST_RecCtrl ://纠偏系统
STRUCT
    Cmd        :ST_RecCmd;
    Io            :ST_RecIo;
    Status      :ST_RecStatus;
END_STRUCT
END_TYPE

// ---- DUTs/04_Rectify/ST_RecCmd.TcDUT
TYPE ST_RecCmd ://纠偏系统
STRUCT
    bLock:				BOOL;	//纠偏外部锁定
	bAuto:				BOOL;	//纠偏自动
	bManual:           BOOL;  //纠偏手动
	bCentre:           BOOL;	//纠偏居中

END_STRUCT
END_TYPE

// ---- DUTs/04_Rectify/ST_RecIo.TcDUT
TYPE ST_RecIo ://纠偏系统
STRUCT
	biAutoDone:				BOOL;	//纠偏自动状态
	biAlarm:           BOOL;	//纠偏故障 

	
    boLock:				BOOL;	//纠偏外部锁定触发
	boAuto:				BOOL;	//纠偏自动切换触发
	boManual:           BOOL;  //纠偏手动切换触发
	boCentre:           BOOL;	//纠偏居中触发

END_STRUCT
END_TYPE

// ---- DUTs/04_Rectify/ST_RecStatus.TcDUT
TYPE ST_RecStatus ://纠偏系统
STRUCT
    bError             :BOOL;     //纠偏故障
    bRuning           :BOOL;    //纠偏运行中
END_STRUCT
END_TYPE

// ---- DUTs/06_Interface/FB_Interface/ST_Cam.TcDUT
TYPE ST_Cam :  //张力FB 接口信号
STRUCT
   	bCamInExecute			                 :BOOL;	
   	bCreatTable		                         :BOOL;	

    bCreatTableDone                        :BOOL;
    bCreatTableError                        :BOOL;
	bError                                       :BOOL;

	bReady                                      :BOOL;
	bStartSync		                             :BOOL;
	bInSync		                                 :BOOL;//同步状态

END_STRUCT
END_TYPE

// ---- DUTs/06_Interface/FB_Interface/ST_Gear.TcDUT
TYPE ST_Gear : //
STRUCT
	bEnable		                        :BOOL;	
	bGearOutMode                 :BOOL;
 
	bReady                            :BOOL;  
	bInGear		 	                   :BOOL;	
	bError				               :BOOL;			
END_STRUCT
END_TYPE

// ---- DUTs/06_Interface/FB_Interface/ST_GearInPos.TcDUT
TYPE ST_GearInPos : //
STRUCT
	bEnable		                        :BOOL;	
   	bEnable2                       :BOOL;	

